(* CoDeSys 2.3 project: drillMachine_v5_WithPackML.pro *)
(* Title: Use of different IEC-61131-3 languages *)
(* Version: 1.0.0 *)
(* Author: Niko Siltala (TUT) *)
(* Description: Use of different IEC-61131-3 languages to control a lift door. *)
(* Libraries: Util.lib 29.1.20 23:45:11, STANDARD.LIB 16.8.17 14:08:57 *)

(* Global variable list: Global_Variables *)
VAR_GLOBAL
	(*Math constants*)
	MATH 				: CONSTANTS_MATH;		(*Mathematical constants from OSCAT 333*)
	lastRandom			: REAL;		(*Last Random number*)

	(*ConveyourIn - Left*)
	I_ConvIn_PartPresent: BOOL;	(*Sensor: Part is present*)
	O_ConvIn_MotON		: BOOL;	(*Conveyour In: Motor ON*)

	(*ConveyourOut - Right*)
	I_ConvOut_PartPresent: BOOL;(*Sensor: Part is present*)
	O_ConvOut_MotON		: BOOL;	(*Conveyour Out: Motor ON*)

	(*Manipulator - Left*)
	I_ManiL_Limit_Up	: BOOL;	(*Manipulator Left: Limit: Up*)
	I_ManiL_Limit_Dn	: BOOL;	(*Manipulator Left: Limit: Down*)
	I_ManiL_Limit_Home	: BOOL;	(*Manipulator Left: Home sensor*)
	I_ManiL_Turned_Left	: BOOL;	(*Manipulator Left: Turned to left*)
	I_ManiL_Turned_Right: BOOL;	(*Manipulator Left: Turned to right*)
	I_ManiL_Gripper_Open: BOOL;	(*Manipulator Left: Gripper is open*)

	O_ManiL_Turn_Left	: BOOL;	(*Manipulator Left: Turn to left position. Controls the valve*)
	O_ManiL_Turn_Right	: BOOL;	(*Manipulator Left: Turn to right position. Controls the valve*)
	O_ManiL_Gripper_Close: BOOL;(*Manipulator Left: Closes Gripper. Controls the valve*)

	bManiL_axZ_Enable	: BOOL;	(*Manipulator Left: Z-axis: enable*)
	bManiL_axZ_Start	: BOOL;	(*Manipulator Left: Z-axis: Start motion*)
	fManiL_axZ_Velo		: REAL;	(*Manipulator Left: Z-axis: Velocity*)
	fManiL_axZ_TargetPos: REAL;	(*Manipulator Left: Z-axis: Target position*)
	fManiL_axZ_CurrPos	: REAL;	(*Manipulator Left: Z-axis: Current position*)
	bManiL_axZ_InTargetPos	: BOOL;	(*Manipulator Left: Z-axis: Target position is reached*)

	(*Drilling Machine*)
	I_Drill_Limit_Up	: BOOL;	(*Drill: Limit: Up*)
	I_Drill_Limit_Dn	: BOOL;	(*Drill: Limit: Down*)
	I_Drill_Limit_Home	: BOOL;	(*Drill: Home sensor*)
	I_Drill_Fixture_Open: BOOL;	(*Drill: Fixture is open*)
	I_Drill_Fixture_Closed: BOOL;	(*Drill: Fixture is closed*)

	O_Drill_Spindle_On	: BOOL;	(*Drill: Turn on drill spindle.*)
	O_Drill_Fixture_Close: BOOL;(*Drill: Closes Fixture. Controls the valve*)

	bDrill_axZ_Enable	: BOOL;	(*Drill: Z-axis: enable*)
	bDrill_axZ_Start	: BOOL;	(*Drill: Z-axis: Start motion*)
	fDrill_axZ_Velo		: REAL;	(*Drill: Z-axis: Velocity*)
	fDrill_axZ_TargetPos: REAL;	(*Drill: Z-axis: Target position*)
	fDrill_axZ_CurrPos	: REAL;	(*Drill: Z-axis: Current position*)
	bDrill_axZ_InTargetPos	: BOOL;	(*Drill: Z-axis: Target position is reached*)

	(*Manipulator - Right*)
	I_ManiR_Limit_Up	: BOOL;	(*Manipulator Right: Limit: Up*)
	I_ManiR_Limit_Dn	: BOOL;	(*Manipulator Right: Limit: Down*)
	I_ManiR_Limit_Home	: BOOL;	(*Manipulator Right: Home sensor*)
	I_ManiR_Turned_Left	: BOOL;	(*Manipulator Right: Turned to left*)
	I_ManiR_Turned_Right: BOOL;	(*Manipulator Right: Turned to right*)
	I_ManiR_Gripper_Open: BOOL;	(*Manipulator Right: Gripper is open*)

	O_ManiR_Turn_Left	: BOOL;	(*Manipulator Right: Turn to left position. Controls the valve*)
	O_ManiR_Turn_Right	: BOOL;	(*Manipulator Right: Turn to right position. Controls the valve*)
	O_ManiR_Gripper_Close: BOOL;(*Manipulator Right: Closes Gripper. Controls the valve*)

	bManiR_axZ_Enable	: BOOL;	(*Manipulator Right: Z-axis: enable*)
	bManiR_axZ_Start	: BOOL;	(*Manipulator Right: Z-axis: Start motion*)
	fManiR_axZ_Velo		: REAL;	(*Manipulator Right: Z-axis: Velocity*)
	fManiR_axZ_TargetPos: REAL;	(*Manipulator Right: Z-axis: Target position*)
	fManiR_axZ_CurrPos	: REAL;	(*Manipulator Right: Z-axis: Current position*)
	bManiR_axZ_InTargetPos	: BOOL;	(*Manipulator Right: Z-axis: Target position is reached*)


	(*Control panel and indications*)
	I_EmergencyClear	: BOOL;	(*Emergency Circuit is clear*)
	I_Btn_Reset		: BOOL;	(*Button: Reset*)
	I_Btn_Start		: BOOL;	(*Button: Start*)
	I_Btn_Stop		: BOOL;	(*Button: Stop*)

	O_Light_Start	: BOOL;	(*Light: Running*)
	O_Light_Stop	: BOOL;	(*Light: Stopped*)
	O_Beacon_Red	: BOOL;	(*Beacon Light: red*)
	O_Beacon_Yellow	: BOOL;	(*Beacon Light: yellow*)
	O_Beacon_Green	: BOOL;	(*Beacon Light: green*)

(* -------------HMI INPUTS (from HMI to PLC) -------------------*)
	HMI_uModeReq		: UINT :=1;		(*Mode request. DEFAULT:PRODUCTION1*)
(* -------------HMI OUTPUTS (from PLC to HMI) -------------------*)
	PLC_uModeCurrent	: UINT;			(*Current Mode*)
	PLC_uStateCurrent	: UINT;			(*Current State*)

(*-----------------------FUNCTION BLOCKS----------------*)
	fbStateModel		: FB_PackMLStateModel_ST;	(*FB for executing PackML state model*)
END_VAR

(* Data type *)
TYPE CONSTANTS_MATH :
STRUCT
	PI : REAL := 	3.14159265358979323846264338327950288;		(* Kreiszahl PI *)
	PI2 : REAL := 	6.28318530717958647692528676655900576;	(* PI * 2 *)
	PI4 : REAL :=  12.56637061435917295385057353311801152;	(* PI * 4 *)
	PI05 : REAL :=  1.5707963267949;							(* PI / 2 *)
	PI025 : REAL := 0.785398163397448;							(* PI / 4 *)
	PI_INV : REAL := 0.318309886183791;						(* 1 / PI *)
	E : REAL := 	2.71828182845904523536028747135266249;		(* Euler constant e *)
	E_INV : REAL := 0.367879441171442;							(* 1 / e *)
	SQ2 : REAL :=	1.4142135623731;							(* Wurzel von 2 *)
	FACTS : ARRAY[0..12] OF DINT := 1,1,2,6,24,120,720,5040,40320,362880,3628800,39916800,479001600;
END_STRUCT
END_TYPE



(*
From OSCAT 333
revision history
hm	26.10.2008	rev 1.0
	original version

hm	26. mar. 2011	rev 1.1
	added array facts
*)

(* Data type *)
TYPE E_Mode :
(*UserModes: Modes for different production states*)
(
	eMode_undefined := 0,
	eMode_Automatic :=1,
	eMode_Manual :=3,
	eMode_Production1 :=5,
	eMode_Production2 :=6
);
END_TYPE

(* Data type *)
TYPE E_ModeProc :
(*Procedural control modes. Can be changed in any state*)
(
	eModeProc_undefined := 0,
	eModeProc_Automatic :=1,
	eModeProc_SemiAutomatic :=2,
	eModeProc_Manual :=3
);
END_TYPE

(* Data type *)
TYPE E_PackMLState :
(*PackML States*)
(
	eSt_Aborting :=0,
	eSt_Aborted,
	eSt_Clearing,
	eSt_Stopped,
	eSt_Stopping,
	eSt_Resetting,
	eSt_Idle,
	eSt_Starting,
	eSt_Execute,
	eSt_Suspending,
	eSt_Suspended,
	eSt_Unsuspending,
	eSt_Holding,
	eSt_Held,
	eSt_UnHolding,
	eSt_Completing,
	eSt_Completed
);
END_TYPE

(* Data type *)
TYPE EN_Mode :
	(eMode_Unknown := 0,
	eMode_Auto := 1,
	eMode_Manual );
END_TYPE

(* Data type *)
TYPE ST_Part :
(*Data structure for the simulated parts *)
STRUCT
	bExists		: BOOL;	(* Part exists *)
	bHasHole	: BOOL;	(* Part has hole *)
	posX		: REAL;	(* X-position of the part*)
	posY		: REAL;	(* Y-position of the part*)
END_STRUCT
END_TYPE

(* POU PRG/PRG_Blinking, ST *)
PROGRAM PRG_Blinking
(*Avustavia laskentaoperaatioita
- vilkutussignaalit
Author: Niko Siltala, niko.siltala@tut.fi, Tampere University of Technology / MEI
Date: 2016-12-12
Version: 1.0
*)
VAR_OUTPUT
	bSign4Hz:BOOL;					(*4 Hz (240krt/min) taajudella vaihteleva signaali*)
	bSign2Hz:BOOL;					(*2 Hz (120krt/min) taajudella vaihteleva signaali*)
	bSign1Hz:BOOL;					(*1 Hz (60krt/min) taajudella vaihteleva signaali*)
	bSign0_5Hz:BOOL;				(*0,5 Hz (30krt/min) taajudella vaihteleva signaali*)
END_VAR
VAR
	bInitDone	: BOOL	:=FALSE;	(*Ohjelman initialisointi*)
	TP_Delay:TP;				(*Nopein taajuus / 2 tuottaja*)
	bBaseHz:BOOL:=FALSE;		(*Nopein taajuus/2*)
	iBaseHz:UINT:=4;				(*Base taajuus (Hz)*)
	(*RTRIG_BASE: R_TRIG;		(*Base signaali nousee*)*)
	RTRIG_2Hz_Sign : R_TRIG;		(*2Hz signaalin generointi*)
	RTRIG_1Hz_Sign : R_TRIG;		(*1Hz signaalin generointi*)
	RTRIG_0_5Hz_Sign : R_TRIG;	(*0,5Hz signaalin generointi*)
	tBaseTaajuus:TIME;			(*Base vilkutuksen timerin arvo. f/2*)
	fPLC_CYCLE_TIME: LREAL;	(*PLC:n cycli aika. Sekunttia*)

END_VAR
(*Ohjelman initialisoinnit - Suoritetaan vain kertaalleen*)
IF NOT bInitDone THEN
	(*fPLC_CYCLE_TIME := UDINT_TO_LREAL(SystemTaskInfoArr[1].cycleTime) / 10E6; (*[s]*)*)
	fPLC_Cycle_Time := 1;	(*[s]*)
	(*Base Vilkkusignaalien tuottaminen*)
	(* 250ms - 1* cykliaika(20ms)*)
	tBaseTaajuus := LREAL_TO_TIME( ( (1/ UINT_TO_LREAL(iBaseHz) / 2 ) - 1 * fPLC_CYCLE_TIME ) * 1000);
	bInitDone := TRUE;
END_IF;

(*Base signaalin genrointi*)
TP_Delay(IN:=NOT TP_Delay.Q , PT:=tBaseTaajuus);
IF NOT TP_Delay.Q THEN
	bBaseHz := NOT bBaseHz;
	bSign4Hz:= bBaseHz;
END_IF;

(*2Hz signaalin genrointi*)
RTRIG_2Hz_Sign(CLK:=bSign4Hz);
IF RTRIG_2Hz_Sign.Q THEN
	bSign2Hz:=NOT bSign2Hz;
END_IF;

(*1Hz signaalin genrointi*)
RTRIG_1Hz_Sign(CLK:=bSign2Hz);
IF RTRIG_1Hz_Sign.Q THEN
	bSign1Hz:=NOT bSign1Hz;
END_IF;

(*0,5 Hz signaalin generointi*)
RTRIG_0_5Hz_Sign(CLK:=bSign1Hz);
IF (RTRIG_0_5Hz_Sign.Q) THEN
	bSign0_5Hz:= NOT bSign0_5Hz;
END_IF;
END_PROGRAM

(* POU PRG/PRG_ConveyorL, ST *)
PROGRAM PRG_ConveyorL
VAR_INPUT
	(* PackML Inputs *)
	State							: E_PackMLState;
	ControlMode					: E_Mode;
	ProceeduralMode				: E_ModeProc;

	hiPartAvail_FromLeft			: BOOL;
	hiRdyToReceive_FromRight  : BOOL;
END_VAR
VAR_OUTPUT
	(* PackML Outputs *)
	SC								: BOOL;
	bInitDone						: BOOL;
	bStopOk						: BOOL;
	bSuspend						: BOOL;

	hoReadyToRecieve_ToLeft	: BOOL;
	hoPartAvail_ToRight			: BOOL;
END_VAR
VAR
	initOK							: BOOL := FALSE;
	fbConveyorLeft				: FB_Conveyor_Left;
END_VAR
SC := FALSE;

CASE State OF
	eSt_Aborting:
		O_ConvIn_MotON		:= FALSE;
		SC 					:= TRUE;
	eSt_Clearing:
		SC 					:= TRUE;
	eSt_Resetting:
		SC 					:= TRUE;
	eSt_Starting:
		SC 					:= TRUE;
	;
	eSt_Holding:
	;
	eSt_UnHolding:
	;
	eSt_Suspending:
		fbConveyorLeft (I_Enable :=  FALSE);
		actUpdateIO;
		IF fbConveyorLeft.bStopOk THEN
			SC := TRUE;
		END_IF
	;
	eSt_Suspended:
		actUpdateIO;
		IF NOT fbConveyorLeft.bSuspend THEN
			bSuspend := FALSE;
		END_IF

	eSt_Unsuspending:
		SC := TRUE;
	eSt_Execute:
		CASE ControlMode OF
			eMode_Automatic:
				fbConveyorLeft (I_Enable	:= TRUE ,	I_Reset := FALSE );
				actUpdateIO;
				IF fbConveyorLeft.bSuspend THEN
					bSuspend := TRUE;
				ELSE
					bSuspend := FALSE;
				END_IF
			eMode_Manual:
			;
		END_CASE
		eSt_Completing:
		;

		eSt_Stopping:
			fbConveyorLeft (I_Enable :=  FALSE);
			actUpdateIO;
			IF fbConveyorLeft.bStopOk THEN
				bStopOk := TRUE;
				SC 	   := TRUE;
			ELSE
				bStopOk := FALSE;
			END_IF
END_CASE
END_PROGRAM
ACTION actUpdateIO:
fbConveyorLeft (
	I_PartEndSensor				:=  I_ConvIn_PartPresent,
	O_ConvRunning				=> O_ConvIn_MotON,
	hiPartAvail_FromLeft			:= hiPartAvail_FromLeft ,
	hiRdyToReceive_FromRight	:= hiRdyToReceive_FromRight,
	hoPartAvail_toRight			=> hoPartAvail_ToRight ,
	hoReadyToRecieve_ToLeft	=> hoReadyToRecieve_ToLeft );
END_ACTION

(* POU FBs/FB_Conveyor_Left, SFC *)
FUNCTION_BLOCK FB_Conveyor_Left
VAR_INPUT
	(* PackML Inputs *)
	State							: E_PackMLState;
	ControlMode					: E_Mode;
	ProceeduralMode				: E_ModeProc;

	I_Enable		 				: BOOL;
	I_Reset		 				: BOOL;
	I_PartEndSensor 				: BOOL;

	(* SMEMA Handshake Inputs *)
	hiPartAvail_FromLeft			: BOOL;
	hiRdyToReceive_FromRight	: BOOL;
END_VAR
VAR_OUTPUT
	(* PackML Outputs *)
	SC								: BOOL;

	(* SMEMA Handshake Outputs *)
	hoReadyToRecieve_ToLeft	: BOOL;
	hoPartAvail_ToRight			: BOOL;

	bInitialised					: BOOL;
	O_ConvRunning			       : BOOL;
	bStopOk						: BOOL;
	bSuspend						: BOOL;

END_VAR
VAR
	tonSuspendDelay			: TON;
	tSuspendDelay			: TIME := T#5s;
	bStartTrans				: BOOL := FALSE;
	bStopTrans				: BOOL := FALSE;
	bTranFinished			: BOOL := FALSE;
	bMachineReady			: BOOL := FALSE;
	bLocalReset				: BOOL := FALSE;	(*Performs local reset*)
	SFCReset 				: BOOL := FALSE;	(*Resets the execution of SFC to init once this SFCFlag is set true *)
END_VAR
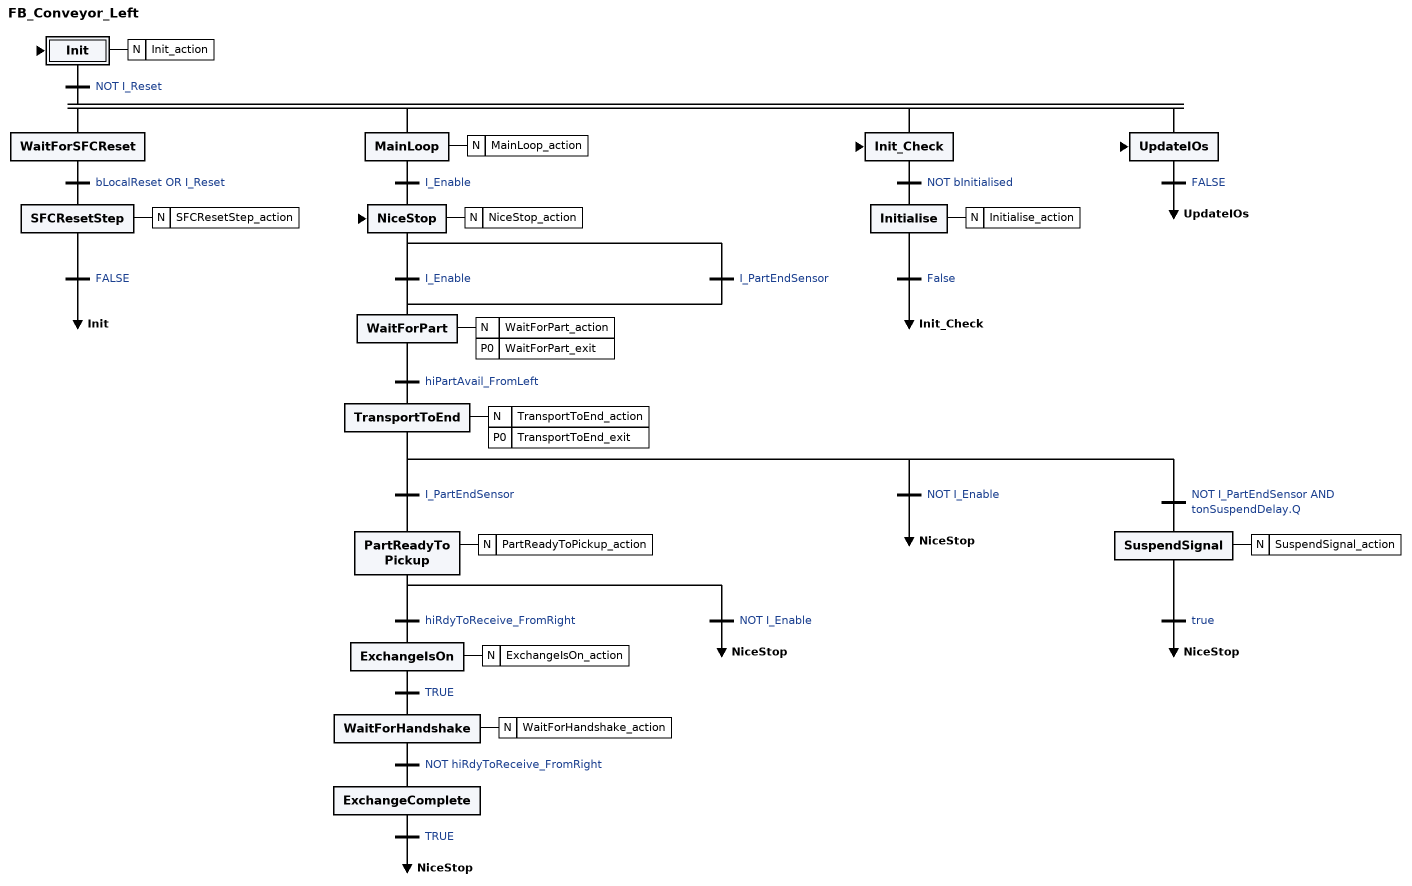
INITIAL_STEP Init:
	Init_action(N);
END_STEP
TRANSITION FROM Init TO (WaitForSFCReset, MainLoop, Init_Check, UpdateIOs) := NOT I_Reset;
END_TRANSITION
STEP WaitForSFCReset:
END_STEP
TRANSITION FROM WaitForSFCReset TO SFCResetStep := bLocalReset OR I_Reset;
END_TRANSITION
STEP MainLoop:
	MainLoop_action(N);
END_STEP
TRANSITION FROM MainLoop TO NiceStop := I_Enable;
END_TRANSITION
STEP Init_Check:
END_STEP
TRANSITION FROM Init_Check TO Initialise := NOT bInitialised;
END_TRANSITION
STEP Initialise:
	Initialise_action(N);
END_STEP
TRANSITION FROM Initialise TO Init_Check := False;
END_TRANSITION
STEP NiceStop:
	NiceStop_action(N);
END_STEP
TRANSITION FROM NiceStop TO WaitForPart := I_Enable;
END_TRANSITION
TRANSITION FROM NiceStop TO WaitForPart := I_PartEndSensor;
END_TRANSITION
STEP WaitForPart:
	WaitForPart_action(N);
	WaitForPart_exit(P0);
END_STEP
TRANSITION FROM WaitForPart TO TransportToEnd := hiPartAvail_FromLeft;
END_TRANSITION
STEP TransportToEnd:
	TransportToEnd_action(N);
	TransportToEnd_exit(P0);
END_STEP
TRANSITION FROM TransportToEnd TO PartReadyToPickup := I_PartEndSensor;
END_TRANSITION
TRANSITION FROM TransportToEnd TO NiceStop := NOT I_Enable;
END_TRANSITION
TRANSITION FROM TransportToEnd TO SuspendSignal := NOT I_PartEndSensor AND tonSuspendDelay.Q;
END_TRANSITION
STEP SuspendSignal:
	SuspendSignal_action(N);
END_STEP
TRANSITION FROM SuspendSignal TO NiceStop := true;
END_TRANSITION
STEP PartReadyToPickup:
	PartReadyToPickup_action(N);
END_STEP
TRANSITION FROM PartReadyToPickup TO ExchangeIsOn := hiRdyToReceive_FromRight;
END_TRANSITION
TRANSITION FROM PartReadyToPickup TO NiceStop := NOT I_Enable;
END_TRANSITION
STEP ExchangeIsOn:
	ExchangeIsOn_action(N);
END_STEP
TRANSITION FROM ExchangeIsOn TO WaitForHandshake := TRUE;
END_TRANSITION
STEP WaitForHandshake:
	WaitForHandshake_action(N);
END_STEP
TRANSITION FROM WaitForHandshake TO ExchangeComplete := NOT hiRdyToReceive_FromRight;
END_TRANSITION
STEP ExchangeComplete:
END_STEP
TRANSITION FROM ExchangeComplete TO NiceStop := TRUE;
END_TRANSITION
STEP UpdateIOs:
END_STEP
TRANSITION FROM UpdateIOs TO UpdateIOs := FALSE;
END_TRANSITION
STEP SFCResetStep:
	SFCResetStep_action(N);
END_STEP
TRANSITION FROM SFCResetStep TO Init := FALSE;
END_TRANSITION

ACTION Init_action:
SFCReset 		:= FALSE;
bLocalReset		:= FALSE;
O_ConvRunning	:= FALSE;
bStopOk 			:= TRUE;
bInitialised		:= FALSE;
bSuspend	 		:= FALSE;
END_ACTION

ACTION MainLoop_action:
hoPartAvail_toRight := FALSE;
END_ACTION

ACTION Initialise_action:
bInitialised := TRUE;
END_ACTION

ACTION NiceStop_action:
bStopOk := TRUE;
O_ConvRunning := TRUE;
hoPartAvail_ToRight := FALSE;
END_ACTION

ACTION WaitForPart_action:
hoReadyToRecieve_ToLeft := TRUE;
bSuspend	 := FALSE;
END_ACTION

ACTION WaitForPart_exit:
bStopOk := FALSE;
END_ACTION

ACTION TransportToEnd_action:
O_ConvRunning := TRUE;
tonSuspendDelay(IN:=TRUE , PT:= tSuspendDelay);
END_ACTION

ACTION TransportToEnd_exit:
tonSuspendDelay(IN:=FALSE);
END_ACTION

ACTION SuspendSignal_action:
bSuspend := TRUE;
END_ACTION

ACTION PartReadyToPickup_action:
hoPartAvail_ToRight := TRUE;
END_ACTION

ACTION ExchangeIsOn_action:
hoReadyToRecieve_ToLeft := FALSE;
END_ACTION

ACTION WaitForHandshake_action:
hoPartAvail_ToRight := FALSE;
END_ACTION

ACTION SFCResetStep_action:
SFCReset := TRUE;
END_ACTION
END_FUNCTION_BLOCK

(* POU PRG/PRG_ConveyorR, ST *)
PROGRAM PRG_ConveyorR
VAR_INPUT
	(* PackML Inputs *)
	State							: E_PackMLState;
	ControlMode					: E_Mode;
	ProceeduralMode				: E_ModeProc;

	hiPartAvail_FromLeft			: BOOL;
	hiRdyToReceive_FromRight  : BOOL;
END_VAR
VAR_OUTPUT
	(* PackML Outputs *)
	SC								: BOOL;
	bInitDone						: BOOL;
	bStopOk						: BOOL;

	hoReadyToRecieve_ToLeft	: BOOL;
	hoPartAvail_ToRight			: BOOL;
END_VAR
VAR
	initOK							: BOOL := FALSE;
	fbConveyorRight				: FB_Conveyor_Right;
END_VAR
SC := FALSE;

CASE State OF
	eSt_Aborting:
		O_ConvOut_MotON		:= FALSE;
		SC := TRUE;
	eSt_Clearing:
		SC := TRUE;
	eSt_Resetting:
		SC := TRUE;
	eSt_Starting:
		SC  := TRUE;
	eSt_Holding:
	;
	eSt_UnHolding:
	;
	eSt_Suspending:
		fbConveyorRight (I_Enable :=  FALSE);
		actUpdateIO;
		IF fbConveyorRight.bStopOk THEN
			SC := TRUE;
		END_IF
	eSt_Unsuspending:
		SC := TRUE;
	eSt_Execute:
		CASE ControlMode OF
			eMode_Automatic:
				fbConveyorRight (I_Enable := TRUE , I_Reset := FALSE );
				actUpdateIO;
			eMode_Manual:
			;
		END_CASE
	eSt_Completing:
	;

	eSt_Stopping:
		fbConveyorRight (I_Enable :=  FALSE);
		actUpdateIO;
		IF fbConveyorRight.bStopOk THEN
			bStopOk := TRUE;
			SC 	   := TRUE;
		ELSE
			bStopOk := FALSE;
			END_IF
END_CASE
END_PROGRAM
ACTION actUpdateIO:
fbConveyorRight (
	I_PartEndSensor				:=  I_ConvOut_PartPresent,
	O_ConvRunning				=> O_ConvOut_MotON,
	hiPartAvail_FromLeft			:= hiPartAvail_FromLeft ,
	hiRdyToReceive_FromRight	:= hiRdyToReceive_FromRight,
	hoPartAvail_toRight			=> hoPartAvail_ToRight ,
	hoReadyToRecieve_ToLeft	=> hoReadyToRecieve_ToLeft );
END_ACTION

(* POU FBs/FB_Conveyor_Right, SFC *)
FUNCTION_BLOCK FB_Conveyor_Right
VAR_INPUT
	(* PackML Inputs *)
	State							: E_PackMLState;
	ControlMode					: E_Mode;
	ProceeduralMode				: E_ModeProc;

	I_Enable		 				: BOOL;
	I_Reset		 				: BOOL;
	I_PartEndSensor 				: BOOL;

	(* SMEMA Handshake Inputs *)
	hiPartAvail_FromLeft			: BOOL;
	hiRdyToReceive_FromRight	: BOOL;
END_VAR
VAR_OUTPUT
	(* PackML Outputs *)
	SC								: BOOL;

	(* SMEMA Handshake Outputs *)
	hoReadyToRecieve_ToLeft	: BOOL;
	hoPartAvail_ToRight			: BOOL;
	O_ConvRunning			       : BOOL;
	bInitialised					: BOOL;
	bStopOk						: BOOL;


END_VAR
VAR
	bStartTrans				: BOOL := FALSE;
	bStopTrans				: BOOL := FALSE;
	bTranFinished			: BOOL := FALSE;
	bMachineReady			: BOOL := FALSE;
	bLocalReset				: BOOL := FALSE;	(*Performs local reset*)
	SFCReset 				: BOOL := FALSE;	(*Resets the execution of SFC to init once this SFCFlag is set true *)
	I_Sensor_PartInsideMachine: BOOL;
END_VAR
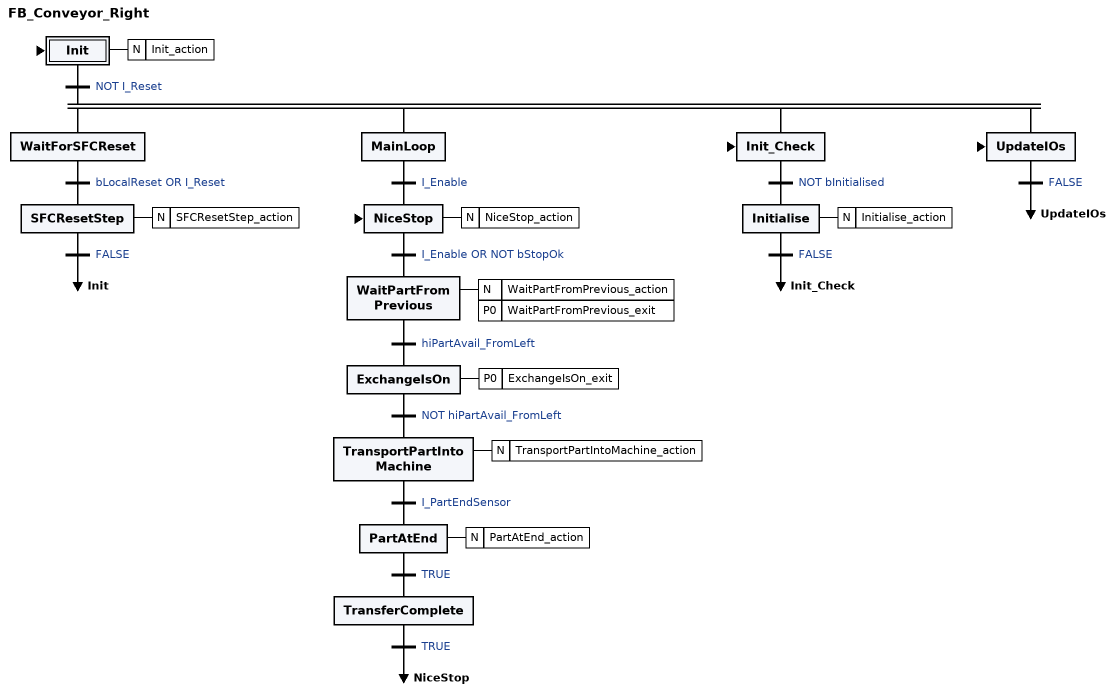
INITIAL_STEP Init:
	Init_action(N);
END_STEP
TRANSITION FROM Init TO (WaitForSFCReset, MainLoop, Init_Check, UpdateIOs) := NOT I_Reset;
END_TRANSITION
STEP WaitForSFCReset:
END_STEP
TRANSITION FROM WaitForSFCReset TO SFCResetStep := bLocalReset OR I_Reset;
END_TRANSITION
STEP MainLoop:
END_STEP
TRANSITION FROM MainLoop TO NiceStop := I_Enable;
END_TRANSITION
STEP Init_Check:
END_STEP
TRANSITION FROM Init_Check TO Initialise := NOT bInitialised;
END_TRANSITION
STEP Initialise:
	Initialise_action(N);
END_STEP
TRANSITION FROM Initialise TO Init_Check := FALSE;
END_TRANSITION
STEP NiceStop:
	NiceStop_action(N);
END_STEP
TRANSITION FROM NiceStop TO WaitPartFromPrevious := I_Enable OR NOT bStopOk;
END_TRANSITION
STEP WaitPartFromPrevious:
	WaitPartFromPrevious_action(N);
	WaitPartFromPrevious_exit(P0);
END_STEP
TRANSITION FROM WaitPartFromPrevious TO ExchangeIsOn := hiPartAvail_FromLeft;
END_TRANSITION
STEP ExchangeIsOn:
	ExchangeIsOn_exit(P0);
END_STEP
TRANSITION FROM ExchangeIsOn TO TransportPartIntoMachine := NOT hiPartAvail_FromLeft;
END_TRANSITION
STEP TransportPartIntoMachine:
	TransportPartIntoMachine_action(N);
END_STEP
TRANSITION FROM TransportPartIntoMachine TO PartAtEnd := I_PartEndSensor;
END_TRANSITION
STEP PartAtEnd:
	PartAtEnd_action(N);
END_STEP
TRANSITION FROM PartAtEnd TO TransferComplete := TRUE;
END_TRANSITION
STEP TransferComplete:
END_STEP
TRANSITION FROM TransferComplete TO NiceStop := TRUE;
END_TRANSITION
STEP UpdateIOs:
END_STEP
TRANSITION FROM UpdateIOs TO UpdateIOs := FALSE;
END_TRANSITION
STEP SFCResetStep:
	SFCResetStep_action(N);
END_STEP
TRANSITION FROM SFCResetStep TO Init := FALSE;
END_TRANSITION

ACTION Init_action:
SFCReset := FALSE;
bLocalReset	:= FALSE;
O_ConvRunning := FALSE;
bStopOK	 := TRUE;
bInitialised := FALSE;
END_ACTION

ACTION Initialise_action:
bInitialised := TRUE;
END_ACTION

ACTION NiceStop_action:
IF hiPartAvail_FromLeft THEN
	bStopOk := FALSE;
ELSE
	bStopOk := TRUE;
END_IF
END_ACTION

ACTION WaitPartFromPrevious_action:
hoReadyToRecieve_ToLeft := TRUE;
hoPartAvail_toRight := FALSE;
END_ACTION

ACTION WaitPartFromPrevious_exit:
bStopOK	:= FALSE;
END_ACTION

ACTION ExchangeIsOn_exit:
O_ConvRunning := FALSE;
END_ACTION

ACTION TransportPartIntoMachine_action:
O_ConvRunning := TRUE;
hoReadyToRecieve_ToLeft := FALSE;
END_ACTION

ACTION PartAtEnd_action:
O_ConvRunning := FALSE;
hoPartAvail_ToRight := TRUE;
END_ACTION

ACTION SFCResetStep_action:
SFCReset := TRUE;
END_ACTION
END_FUNCTION_BLOCK

(* POU PRG/PRG_Drill, ST *)
PROGRAM PRG_Drill
VAR_INPUT
	(* PackML Inputs *)
	State							: E_PackMLState;
	ControlMode					: E_Mode;
	ProceeduralMode				: E_ModeProc;

	hiPartAvail_FromLeft			: BOOL;
	hiRdyToReceive_FromRight  : BOOL;
END_VAR
VAR_OUTPUT
	(* PackML Outputs *)
	SC								: BOOL;
	bInitDone						: BOOL;
	bStopOk						: BOOL;

	hoReadyToRecieve_ToLeft	: BOOL;
	hoPartAvail_ToRight			: BOOL;
END_VAR
VAR
	fbDrill 							: FB_Drill;
END_VAR
SC := FALSE;

CASE State OF
	eSt_Aborting:
		bDrill_axZ_Start 					:= FALSE;
		O_Drill_Spindle_On				:= FALSE;
		(*  Avoid Toggling fixture Objects *)
		IF I_Drill_Fixture_Open THEN
			O_Drill_Fixture_Close 		:= FALSE;
		ELSE
			O_Drill_Fixture_Close		:= TRUE;
		END_IF
		SC := TRUE;
	eSt_Clearing:
		SC := TRUE;
	eSt_Resetting:
		SC := TRUE;
	eSt_Starting:
		IF NOT  fbDrill.bInitialised THEN
			actUpdateIO;
		ELSE
			bInitDone	 := TRUE;
			SC		 := TRUE;
		END_IF

	;
	eSt_Holding:
	;
	eSt_UnHolding:
	;
	eSt_Suspending:
		fbDrill (I_Enable :=  FALSE);
		actUpdateIO;
		IF fbDrill.bStopOk THEN
			SC := TRUE;
		END_IF
	eSt_Unsuspending:
		SC := TRUE;
	eSt_Execute:
		CASE ControlMode OF
			eMode_Automatic:
				fbDrill (
					I_Enable						:= TRUE,
					I_Reset						:= FALSE);
				actUpdateIO;
			eMode_Manual:
			;
		END_CASE
		eSt_Completing:
		;

		eSt_Stopping:
			fbDrill (I_Enable :=  FALSE);
			actUpdateIO;
			IF fbDrill.bStopOk THEN
				bStopOk := TRUE;
				SC 	   := TRUE;
			ELSE
				bStopOk := FALSE;
			END_IF
END_CASE
END_PROGRAM
ACTION actUpdateIO:
fbDrill (
	I_Drill_Limit_Up				:= I_Drill_Limit_Up,
	I_Drill_Limit_Dn				:= I_Drill_Limit_Dn ,
	I_Drill_Limit_Home			:= I_Drill_Limit_Home,
	I_Drill_Fixture_Open			:= I_Drill_Fixture_Open,
	I_Drill_Fixture_Closed		:= I_Drill_Fixture_Closed,
	fDrill_axZ_CurrPos			:= fDrill_axZ_CurrPos ,
	bDrill_axZ_InTargetPos		:= bDrill_axZ_InTargetPos ,

	hiPartAvail_FromLeft			:= hiPartAvail_FromLeft ,
	hiRdyToReceive_FromRight	:= hiRdyToReceive_FromRight ,
	hoReadyToRecieve_ToLeft	=>hoReadyToRecieve_ToLeft ,
	hoPartAvail_ToRight			=>hoPartAvail_ToRight ,

	O_Drill_Spindle_On			=> O_Drill_Spindle_On ,
	O_Drill_Fixture_Close		=> O_Drill_Fixture_Close ,
	bDrill_axZ_Enable			=> bDrill_axZ_Enable ,
	bDrill_axZ_Start				=> bDrill_axZ_Start ,
	fDrill_axZ_Velo				=> fDrill_axZ_Velo,
	fDrill_axZ_TargetPos			=> fDrill_axZ_TargetPos );
END_ACTION

(* POU FBs/FB_Drill, SFC *)
FUNCTION_BLOCK FB_Drill
VAR_INPUT
	(* PackML Inputs *)
	State							: E_PackMLState;
	ControlMode					: E_Mode;
	ProceeduralMode				: E_ModeProc;

	I_Enable		 				: BOOL;
	I_Reset		 				: BOOL;
	I_StopRequest				: BOOL;

	(* SMEMA HandshakeInputs *)
	hiPartAvail_FromLeft			: BOOL;
	hiRdyToReceive_FromRight	: BOOL;

	(* Drill Sensor *)
	I_Drill_Limit_Up				: BOOL;	(*Drill: Limit: Up*)
	I_Drill_Limit_Dn				: BOOL;	(*Drill: Limit: Down*)
	I_Drill_Limit_Home			: BOOL;	(*Drill: Home sensor*)
	I_Drill_Fixture_Open			: BOOL;	(*Drill: Fixture is open*)
	I_Drill_Fixture_Closed		: BOOL;	(*Drill: Fixture is closed*)

	(* Drill Inputs Controls *)
	fDrill_axZ_CurrPos			: REAL;	(*Drill: Z-axis: Current position*)
	bDrill_axZ_InTargetPos		: BOOL;	(*Drill: Z-axis: Target position is reached*)
END_VAR
VAR_OUTPUT
	(* PackML Outputs *)
	SC								: BOOL;

	O_Drill_Spindle_On			: BOOL;	(*Drill: Turn on drill spindle.*)
	O_Drill_Fixture_Close		: BOOL;	(*Drill: Closes Fixture. Controls the valve*)
	bInitialised					: BOOL;
	bStopOk						: BOOL;

	(* SMEMA HandshakeInputs *)
	hoReadyToRecieve_ToLeft	: BOOL;
	hoPartAvail_ToRight			: BOOL;

	(* Drill Outputs *)
	bDrill_axZ_Enable			: BOOL;	(*Drill: Z-axis: enable*)
	bDrill_axZ_Start				: BOOL;	(*Drill: Z-axis: Start motion*)
	fDrill_axZ_Velo				: REAL;	(*Drill: Z-axis: Velocity*)
	fDrill_axZ_TargetPos			: REAL;	(*Drill: Z-axis: Target position*)

END_VAR
VAR

	bDrillHomed				: BOOL := FALSE;
	bStartCycle				: BOOL := FALSE;
	bLocalReset				: BOOL := FALSE;	(*Performs local reset*)
	SFCReset 				: BOOL := FALSE;	(*Resets the execution of SFC to init once this SFCFlag is set true *)
	tonMoveDelay				: TON;
	tMoveDelay				: TIME := T#1s;
	bDrill						: BOOL;
	bDrilled					: BOOL;

END_VAR
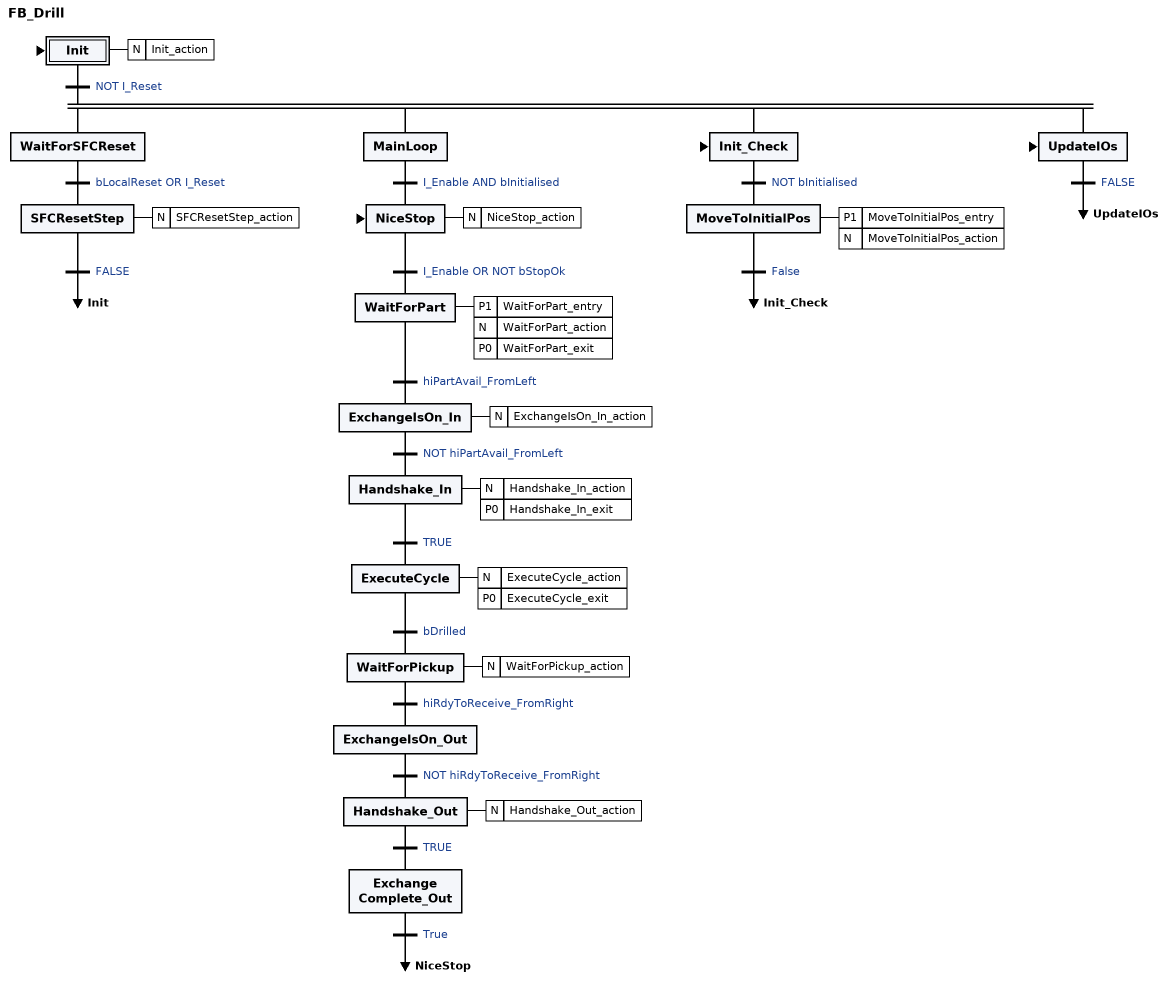
INITIAL_STEP Init:
	Init_action(N);
END_STEP
TRANSITION FROM Init TO (WaitForSFCReset, MainLoop, Init_Check, UpdateIOs) := NOT I_Reset;
END_TRANSITION
STEP WaitForSFCReset:
END_STEP
TRANSITION FROM WaitForSFCReset TO SFCResetStep := bLocalReset OR I_Reset;
END_TRANSITION
STEP MainLoop:
END_STEP
TRANSITION FROM MainLoop TO NiceStop := I_Enable AND bInitialised;
END_TRANSITION
STEP Init_Check:
END_STEP
TRANSITION FROM Init_Check TO MoveToInitialPos := NOT bInitialised;
END_TRANSITION
STEP MoveToInitialPos:
	MoveToInitialPos_entry(P1);
	MoveToInitialPos_action(N);
END_STEP
TRANSITION FROM MoveToInitialPos TO Init_Check := False;
END_TRANSITION
STEP NiceStop:
	NiceStop_action(N);
END_STEP
TRANSITION FROM NiceStop TO WaitForPart := I_Enable OR NOT bStopOk;
END_TRANSITION
STEP WaitForPart:
	WaitForPart_entry(P1);
	WaitForPart_action(N);
	WaitForPart_exit(P0);
END_STEP
TRANSITION FROM WaitForPart TO ExchangeIsOn_In := hiPartAvail_FromLeft;
END_TRANSITION
STEP ExchangeIsOn_In:
	ExchangeIsOn_In_action(N);
END_STEP
TRANSITION FROM ExchangeIsOn_In TO Handshake_In := NOT hiPartAvail_FromLeft;
END_TRANSITION
STEP Handshake_In:
	Handshake_In_action(N);
	Handshake_In_exit(P0);
END_STEP
TRANSITION FROM Handshake_In TO ExecuteCycle := TRUE;
END_TRANSITION
STEP ExecuteCycle:
	ExecuteCycle_action(N);
	ExecuteCycle_exit(P0);
END_STEP
TRANSITION FROM ExecuteCycle TO WaitForPickup := bDrilled;
END_TRANSITION
STEP WaitForPickup:
	WaitForPickup_action(N);
END_STEP
TRANSITION FROM WaitForPickup TO ExchangeIsOn_Out := hiRdyToReceive_FromRight;
END_TRANSITION
STEP ExchangeIsOn_Out:
END_STEP
TRANSITION FROM ExchangeIsOn_Out TO Handshake_Out := NOT hiRdyToReceive_FromRight;
END_TRANSITION
STEP Handshake_Out:
	Handshake_Out_action(N);
END_STEP
TRANSITION FROM Handshake_Out TO ExchangeComplete_Out := TRUE;
END_TRANSITION
STEP ExchangeComplete_Out:
END_STEP
TRANSITION FROM ExchangeComplete_Out TO NiceStop := True;
END_TRANSITION
STEP UpdateIOs:
END_STEP
TRANSITION FROM UpdateIOs TO UpdateIOs := FALSE;
END_TRANSITION
STEP SFCResetStep:
	SFCResetStep_action(N);
END_STEP
TRANSITION FROM SFCResetStep TO Init := FALSE;
END_TRANSITION

ACTION Init_action:
(* Status Flags *)
bStopOK			:= TRUE;
bInitialised 		:= FALSE;
bDrillHomed 		:= FALSE;
(* Reset Flags *)
SFCReset 		:= FALSE;
bLocalReset		:= FALSE;
(* Handshake Flags*)
hoReadyToRecieve_ToLeft	:= FALSE;
hoPartAvail_ToRight			:= FALSE;
END_ACTION

ACTION MoveToInitialPos_entry:
bStopOk := FALSE;
END_ACTION

ACTION MoveToInitialPos_action:
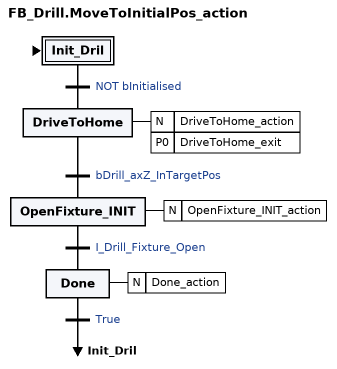
INITIAL_STEP Init_Dril:
END_STEP
TRANSITION FROM Init_Dril TO DriveToHome := NOT bInitialised;
END_TRANSITION
STEP DriveToHome:
	DriveToHome_action(N);
	DriveToHome_exit(P0);
END_STEP
TRANSITION FROM DriveToHome TO OpenFixture_INIT := bDrill_axZ_InTargetPos;
END_TRANSITION
STEP OpenFixture_INIT:
	OpenFixture_INIT_action(N);
END_STEP
TRANSITION FROM OpenFixture_INIT TO Done := I_Drill_Fixture_Open;
END_TRANSITION
STEP Done:
	Done_action(N);
END_STEP
TRANSITION FROM Done TO Init_Dril := True;
END_TRANSITION

ACTION DriveToHome_action:
bDrill_axZ_Enable		:= TRUE;
fDrill_axZ_TargetPos		:= -10;
fDrill_axZ_Velo			:= 5;
bDrill_axZ_Start			:= TRUE;
END_ACTION

ACTION DriveToHome_exit:
bDrill_axZ_Start := FALSE;
END_ACTION

ACTION OpenFixture_INIT_action:
O_Drill_Fixture_Close := FALSE;
END_ACTION

ACTION Done_action:
bInitialised := TRUE;
bStopOk := TRUE;
END_ACTION
END_ACTION

ACTION NiceStop_action:
IF hiPartAvail_FromLeft THEN
	bStopOk := FALSE;
ELSE
	bStopOk := TRUE;
END_IF
END_ACTION

ACTION WaitForPart_entry:
bStopOK	:= TRUE;
END_ACTION

ACTION WaitForPart_action:
hoReadyToRecieve_ToLeft := TRUE;
END_ACTION

ACTION WaitForPart_exit:
bStopOK	:= FALSE;
END_ACTION

ACTION ExchangeIsOn_In_action:
hoReadyToRecieve_ToLeft	:= TRUE;
END_ACTION

ACTION Handshake_In_action:
hoReadyToRecieve_ToLeft := FALSE;
END_ACTION

ACTION Handshake_In_exit:
bDrill := TRUE;
END_ACTION

ACTION ExecuteCycle_action:
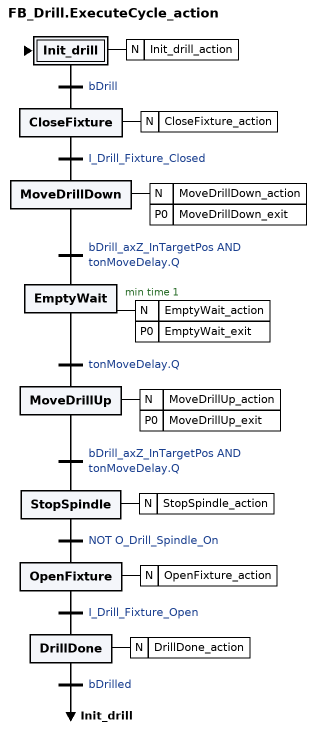
INITIAL_STEP Init_drill:
	Init_drill_action(N);
END_STEP
TRANSITION FROM Init_drill TO CloseFixture := bDrill;
END_TRANSITION
STEP CloseFixture:
	CloseFixture_action(N);
END_STEP
TRANSITION FROM CloseFixture TO MoveDrillDown := I_Drill_Fixture_Closed;
END_TRANSITION
STEP MoveDrillDown:
	MoveDrillDown_action(N);
	MoveDrillDown_exit(P0);
END_STEP
TRANSITION FROM MoveDrillDown TO EmptyWait := bDrill_axZ_InTargetPos AND tonMoveDelay.Q;
END_TRANSITION
STEP EmptyWait: (* min time 1 *)
	EmptyWait_action(N);
	EmptyWait_exit(P0);
END_STEP
TRANSITION FROM EmptyWait TO MoveDrillUp := tonMoveDelay.Q;
END_TRANSITION
STEP MoveDrillUp:
	MoveDrillUp_action(N);
	MoveDrillUp_exit(P0);
END_STEP
TRANSITION FROM MoveDrillUp TO StopSpindle := bDrill_axZ_InTargetPos AND tonMoveDelay.Q;
END_TRANSITION
STEP StopSpindle:
	StopSpindle_action(N);
END_STEP
TRANSITION FROM StopSpindle TO OpenFixture := NOT O_Drill_Spindle_On;
END_TRANSITION
STEP OpenFixture:
	OpenFixture_action(N);
END_STEP
TRANSITION FROM OpenFixture TO DrillDone := I_Drill_Fixture_Open;
END_TRANSITION
STEP DrillDone:
	DrillDone_action(N);
END_STEP
TRANSITION FROM DrillDone TO Init_drill := bDrilled;
END_TRANSITION

ACTION Init_drill_action:
O_Drill_Spindle_On	:= FALSE;
bDrill_axZ_Enable	:= FALSE;
bDrill_axZ_Start		:= FALSE;
fDrill_axZ_Velo		:= 0;
END_ACTION

ACTION CloseFixture_action:
bDrilled 					:= FALSE;
O_Drill_Fixture_Close 	:= TRUE;
END_ACTION

ACTION MoveDrillDown_action:
bDrill_axZ_Enable := TRUE;
fDrill_axZ_Velo :=10;
fDrill_axZ_TargetPos := -140;
bDrill_axZ_Start := TRUE;
tonMoveDelay(IN:=TRUE , PT:= tMoveDelay);
O_Drill_Spindle_On := TRUE;
END_ACTION

ACTION MoveDrillDown_exit:
bDrill_axZ_Start := FALSE;
tonMoveDelay(IN:=FALSE );
END_ACTION

ACTION EmptyWait_action:
tonMoveDelay(IN:=TRUE , PT:= tMoveDelay);
END_ACTION

ACTION EmptyWait_exit:
tonMoveDelay(IN:=FALSE);
END_ACTION

ACTION MoveDrillUp_action:
tonMoveDelay(IN:=TRUE , PT:= tMoveDelay);
fDrill_axZ_Velo :=10;
fDrill_axZ_TargetPos := -10;
bDrill_axZ_Start := TRUE;
END_ACTION

ACTION MoveDrillUp_exit:
bDrill_axZ_Start := FALSE;
tonMoveDelay(IN:=FALSE);
END_ACTION

ACTION StopSpindle_action:
O_Drill_Spindle_On := FALSE;
END_ACTION

ACTION OpenFixture_action:
O_Drill_Fixture_Close	:= FALSE;
END_ACTION

ACTION DrillDone_action:
bDrilled := TRUE;
bDrill := FALSE;
END_ACTION
END_ACTION

ACTION ExecuteCycle_exit:
bDrilled := FALSE;
END_ACTION

ACTION WaitForPickup_action:
hoPartAvail_ToRight := TRUE;
END_ACTION

ACTION Handshake_Out_action:
hoPartAvail_ToRight := FALSE;
END_ACTION

ACTION SFCResetStep_action:
SFCReset := TRUE;
END_ACTION
END_FUNCTION_BLOCK

(* POU PRG_MAIN_DRILL_MACHINE, ST *)
PROGRAM PRG_MAIN_DRILL_MACHINE
VAR
	(* PackML Related Variables *)
	bBlink					: BOOL;	(*1s blinkg for CodeSys Simulation*)
	c						: INT;	(*Support variable for blinking*)

	partCount				: R_TRIG;
	bAllOkToStop		       : BOOL := TRUE;
	bInit_FirstBoot			: BOOL := FALSE;
	bStopRequested		: BOOL := FALSE;
	bE_StopRestart		: BOOL := FALSE;
	oStopRequested		: BOOL;

	itemToProduce 		: INT := 1;
	itemProduced 		: INT := 0;

END_VAR
(* ****** Section 1: Initialisations and default values. Initial conditions for variables on every PLC cycle*)
fbStateModel.bSC := FALSE;
actCountParts;
actCheckOKtoStop;

(* ****** Section 2: Actions in your program without considering the Control Mode. I.e. actions are performed same way indenpendent on
current Control Mode selection.*)
(*Mode independent state actions*)
CASE fbStateModel.eState OF
eSt_Aborting:
	(* One can make specific actions in case of specific Mode-State combination.
	   One can also consider to call a specific program when in specific Mode-State combination*)
	(*actAborting;*)
	bInit_FirstBoot := FALSE;
	fbStateModel.bSC := PRG_ConveyorL.SC AND	PRG_ManipulatorLeft.SC  AND PRG_Drill.SC AND
						     PRG_ManipulatorRight.SC AND  PRG_ConveyorR.SC;
eSt_Clearing:
	fbStateModel.bSC := PRG_ConveyorL.SC AND PRG_ManipulatorLeft.SC  AND PRG_Drill.SC AND
						     PRG_ManipulatorRight.SC AND  PRG_ConveyorR.SC;
eSt_Stopping:
	fbStateModel.bSC := PRG_ConveyorL.SC AND PRG_ManipulatorLeft.SC  AND PRG_Drill.SC AND
						     PRG_ManipulatorRight.SC AND  PRG_ConveyorR.SC;
eSt_Resetting:
	fbStateModel.bSC := PRG_ConveyorL.SC AND PRG_ManipulatorLeft.SC  AND PRG_Drill.SC AND
						     PRG_ManipulatorRight.SC AND  PRG_ConveyorR.SC;
eSt_Holding:
	fbStateModel.bSC := TRUE;		(*TODO: Remove/Replace this row with desired actions*)
eSt_UnHolding:
	fbStateModel.bSC := TRUE;		(*TODO: Remove/Replace this row with desired actions*)
eSt_Suspending:
	fbStateModel.bSC := PRG_ConveyorL.SC AND PRG_ManipulatorLeft.SC  AND PRG_Drill.SC AND
						     PRG_ManipulatorRight.SC AND  PRG_ConveyorR.SC;
	;
	(*fbStateModel.bSC := TRUE; *)		(*TODO: Remove/Replace this row with desired actions*)
eSt_Unsuspending:
	fbStateModel.bSC := PRG_ConveyorL.SC AND PRG_ManipulatorLeft.SC  AND PRG_Drill.SC AND
						     PRG_ManipulatorRight.SC AND  PRG_ConveyorR.SC;
END_CASE;

(* ****** Section 3: Actions in your program which are Control Mode specific. Two nested case structures where outer one selects the
control mode and inner the PackML state. In order to avoid conflicts, it would be better to process each PackML state either in Section 2 
or Section 3, but not in both. *)
(*Execution mode related state actions*)
CASE fbStateModel.eMode OF
(*MODE: MANUAL*)
eMode_Manual:
	(* ****** Section 3.1: PackML state based processing actions when Control Mode is Manual.*)
	CASE fbStateModel.eState OF
	eSt_Idle:
		fbStateModel.bAck_Completed := FALSE;		(*TODO: Remove/Replace this row with desired actions*)
	eSt_Starting:
		fbStateModel.bSC := TRUE;					(*TODO: Remove/Replace this row with desired actions*)
	eSt_Completing:
		fbStateModel.bSC := TRUE;					(*TODO: Remove/Replace this row with desired actions*)
	eSt_Completed:
		fbStateModel.bAck_Completed := TRUE;		(*TODO: Remove/Replace this row with desired actions*)
	END_CASE;

(*MODE: AUTOMATIC*)
eMode_Automatic:
	(* ****** Section 3.2: PackML state based processing actions when Control Mode is Automatic.*)
	CASE fbStateModel.eState OF
	eSt_Idle:
		fbStateModel.bAck_Completed := FALSE;		(*TODO: Remove/Replace this row with desired actions*)
	eSt_Starting:
			fbStateModel.bSC := PRG_ConveyorL.SC AND PRG_ManipulatorLeft.SC  AND PRG_Drill.SC AND
						     		     PRG_ManipulatorRight.SC AND  PRG_ConveyorR.SC;
	eSt_Completing:
		fbStateModel.bSC := TRUE;					(*TODO: Remove/Replace this row with desired actions*)
	eSt_Completed:
		;
		(*fbStateModel.bAck_Completed:= I_Btn_Start;*)
	END_CASE;

(*MODE: UNKNOWN*)
ELSE	(*This is an Error branch.*)
	; (*TODO: Make implementation*)
END_CASE;

(* ****** Section 4: Grouping PackML states for calling Programs or FB instances.
This is to avoid repetition inside case structure in Section 3. With IF clause setting lower (and upper) state limits we can filter out the states when we want to call 
specific programs. The order of states is defined in Tab:Data types > E_PackMLState. eSt_Aborting is lowest and eSt_Completed is highest.
Here we filter calling programs, only when we are in higher states than Stopped. Inside IF there is again CASE which process each Control Mode separately.*)
(*Execution part. Making calls for program if we are on states above Stopped*)
IF (fbStateModel.eState > eSt_Stopped) THEN
	CASE fbStateModel.eMode OF
		(*MODE: MANUAL*)
		eMode_Manual:
			;
		(*MODE: AUTOMATIC*)
		eMode_Automatic:
			;
	END_CASE;
END_IF;

(* ****** Section 5: Calling the fbStateModel instance.
Here the instance of state model is called and all triggering inputs are set, but bSC (State Completed), which you control in your programs. 
This is indication that your program has  finished certain stage.
- Pay attention where the instance fbStateModel is defined. Do you do it in global variables or e.g. here in PRG_MAIN? Important is to use the 
same instance in all places, so that machine state is unique and shared. Remember, if you have multiple definitions, the PRG_MAIN "hides" 
the global one, and might lead to problems elswhere, when you think you are using the same instance, but actually are not. 
- In case you are using the PackML visualisation (VC_PackMLStates), make sure you connect its placeholder to the very same PackML FB instance.
- The Mask for wIgnoreState is created as following. I use binary base for the value(2#). The lowest bit in the mask corresponds the eSt_Aborting
 in E_PackMLState. The next is eSt_Aborted, and so on. Specific state is ignored and jumped over when it is masked out i.e. ignored by having 1 
in that position. Note that implementation allows this only for selected states. See FB_PackMLStateModel_ST code for further details.*)
(*Calling & Updating the state model*)
(*TODO: Evaluate and change all input conditions according your application needs*)
fbStateModel(
	bResetFB			:= ,
	eModeReq		:= HMI_uModeReq,
	wIgnoreState		:= 2#100000,		(*TODO: Which states should be ignodered. Default: 2#000000 or 2#100000*)
	bSC				:= ,		(*Must NOT be assigned ANY variable, because fb input is directly assigned above by your programs!!!*)
	bAbort				:= NOT I_EmergencyClear,
	bClear				:= I_EmergencyClear,
	bReset			:= ,
	bStart				:= I_Btn_Start,
	bHold				:= ,
	bUn_Hold			:= ,
	bSuspend			:= PRG_ConveyorL.bSuspend AND bAllOkToStop,
	bUn_Suspend	:= NOT PRG_ConveyorL.bSuspend,
	bStop				:= I_Btn_Stop,
	bComplete		:= ,
	bAck_Completed	:= ,
	eMode				=> ,
	eState				=> );

(* ****** Section 6: Here we update all outputs according the current state of our PackML model. This allows us to process the in single location.
The control of outputs is bind to state, not e.g. to inputs. The inputs are the one driving the PackML model forward. Again CASE structure can be used.*)
(*Call for HMI and UI update*)
HMI_and_UI_Update;


PRG_ConveyorL(
	State							:= fbStateModel.eState ,
	ControlMode					:= fbStateModel.eMode,
	ProceeduralMode				:= ,
	hiPartAvail_FromLeft			:= TRUE ,
	hiRdyToReceive_FromRight	:= PRG_ManipulatorLeft.hoReadyToRecieve_ToLeft,
	SC								=> ,
	bInitDone						=> ,
	bStopOk						=> ,
	hoReadyToRecieve_ToLeft	=> ,
	hoPartAvail_ToRight			=> );

PRG_ManipulatorLeft(
	State							:= fbStateModel.eState,
	ControlMode					:= fbStateModel.eMode ,
	ProceeduralMode				:= ,
	hiPartAvail_FromLeft			:= PRG_ConveyorL.hoPartAvail_ToRight ,
	hiRdyToReceive_FromRight	:= PRG_Drill.hoReadyToRecieve_ToLeft,
	SC								=> ,
	bInitDone						=> ,
	bStopOk						=> ,
	hoReadyToRecieve_ToLeft	=> ,
	hoPartAvail_ToRight			=> );

PRG_Drill(
	State							:= fbStateModel.eState,
	ControlMode					:= fbStateModel.eMode ,
	ProceeduralMode				:= ,
	hiPartAvail_FromLeft			:= PRG_ManipulatorLeft.hoPartAvail_ToRight ,
	hiRdyToReceive_FromRight	:= PRG_ManipulatorRight.hoReadyToRecieve_ToLeft,
	SC								=> ,
	bInitDone						=> ,
	bStopOk						=> ,
	hoReadyToRecieve_ToLeft	=> ,
	hoPartAvail_ToRight			=> );

PRG_ManipulatorRight(
	State							:= fbStateModel.eState ,
	ControlMode					:= fbStateModel.eMode ,
	ProceeduralMode				:= ,
	hiPartAvail_FromLeft			:= PRG_Drill.hoPartAvail_ToRight,
	hiRdyToReceive_FromRight	:= PRG_ConveyorR.hoReadyToRecieve_ToLeft,
	SC								=> ,
	bInitDone						=> ,
	bStopOk						=> ,
	hoReadyToRecieve_ToLeft	=> ,
	hoPartAvail_ToRight			=> );

PRG_ConveyorR(
	State							:= fbStateModel.eState ,
	ControlMode					:= fbStateModel.eMode,
	ProceeduralMode				:= ,
	hiPartAvail_FromLeft			:= PRG_ManipulatorRight.hoPartAvail_ToRight,
	hiRdyToReceive_FromRight	:= TRUE,
	SC								=> ,
	bInitDone						=> ,
	bStopOk						=> ,
	hoReadyToRecieve_ToLeft	=> ,
	hoPartAvail_ToRight			=> );
END_PROGRAM
ACTION actAborting:
(* Conveyors *)
O_ConvIn_MotON					:= FALSE;
O_ConvOut_MotON	 			:= FALSE;

(* Manipulators *)
O_ManiL_Turn_Left		 		:= FALSE;
O_ManiL_Turn_Right		 		:= FALSE;
O_ManiR_Turn_Left		 		:= FALSE;
O_ManiR_Turn_Right		 		:= FALSE;
bManiL_axZ_Start					:= FALSE;
bManiR_axZ_Start				:= FALSE;

(*  Avoid Dropping Objects *)
IF I_ManiL_Gripper_Open THEN
	O_ManiL_Gripper_Close 	:= FALSE;
ELSE
	O_ManiL_Gripper_Close		:= TRUE;
END_IF
(* Drill *)
bDrill_axZ_Start 					:= FALSE;
O_Drill_Spindle_On				:= FALSE;

(*  Avoid Toggling fixture Objects *)
IF I_Drill_Fixture_Open THEN
	O_Drill_Fixture_Close 		:= FALSE;
ELSE
	O_Drill_Fixture_Close		:= TRUE;
END_IF

(*
fbConveyorLeft(I_Reset:=TRUE, bRun := FALSE);
fbConveyorRight(I_Reset:=TRUE, bRun := FALSE);
fbManipulatorLeft(I_Reset:=TRUE, I_Enable := FALSE);
fbManipulatorRight(I_Reset:=TRUE, I_Enable := FALSE);
fbDrill(I_Reset:=TRUE, I_Enable := FALSE);
*)
END_ACTION
ACTION actCheckOkToStop:
IF PRG_ConveyorL.bStopOk  AND PRG_ManipulatorLeft.bStopOk  AND PRG_Drill.bStopOk AND PRG_ManipulatorRight.bStopOk AND  PRG_ConveyorR.bStopOk THEN
	bAllOkToStop := TRUE;
ELSE
	bAllOkToStop := FALSE;
END_IF
END_ACTION
ACTION actCountParts:
partCount(CLK:= I_ConvOut_PartPresent, Q=> );
IF partCount.Q THEN
	itemProduced := itemProduced + 1;
END_IF
END_ACTION
ACTION HMI_and_UI_Update:
(*HMI Update*)
(*Calling blinking sub-program*)
PRG_Blinking (bSign4Hz=> , bSign2Hz=> , bSign1Hz=> , bSign0_5Hz=> );
(*Codesys simulation 1Hz blinking *)
c:= c + 1;
IF c > 1 THEN
	c:=0;
END_IF;
bBlink := (c=0);	(*bBlink is true if c=0*)

(*Init values*)
O_Light_Stop := FALSE;	(*TODO: Change initial values according your app needs*)

(*TODO: Change values according range of states *)
(*Start light*)
O_Light_Start :=  (fbStateModel.eState > eSt_Idle) AND (fbStateModel.eState < eSt_Completed);
IF (fbStateModel.eState > eSt_Completing) OR (fbStateModel.eState <= eSt_Execute) THEN
	O_Beacon_Yellow := FALSE;
END_IF

CASE fbStateModel.eState OF
eSt_Aborting, eSt_Aborted,eSt_Clearing:
	O_Light_Stop 		 := bBlink;
	O_Beacon_Red 	 := bBlink;
	O_Light_Start 		 := FALSE;
	O_Beacon_Green := FALSE;
eSt_Stopping, eSt_Stopped, eSt_Completed:
	O_Beacon_Green:= FALSE;
	IF  fbStateModel.eState = eSt_Stopping THEN
		O_Beacon_Green:= bBlink;
		O_Light_Start 		:= bBlink;
	END_IF
	O_Light_Stop 		:= TRUE;
	O_Beacon_Red 	:= TRUE;
eSt_Starting:
	O_Light_Start 		:= bBlink;
	O_Light_Stop 		 := FALSE;
	O_Beacon_Green:= bBlink;
	O_Beacon_Red 	 := FALSE;
eSt_Suspended, eSt_Suspending, eSt_Held:
	O_Light_Start 		 := bBlink;
	O_Beacon_Green	 := bBlink;
	O_Beacon_Yellow := TRUE;
	O_Beacon_Red 	 := FALSE;
eSt_Execute:
	O_Beacon_Red 	 := FALSE;
	O_Beacon_Green	 := TRUE;
END_CASE;
END_ACTION

(* POU PRG/PRG_ManipulatorLeft, ST *)
PROGRAM PRG_ManipulatorLeft
VAR_INPUT
	(* PackML Inputs *)
	State							: E_PackMLState;
	ControlMode					: E_Mode;
	ProceeduralMode				: E_ModeProc;

	hiPartAvail_FromLeft			: BOOL;
	hiRdyToReceive_FromRight  : BOOL;
END_VAR
VAR_OUTPUT
	(* PackML Outputs *)
	SC								: BOOL;
	bInitDone						: BOOL;
	bStopOk						: BOOL;

	hoReadyToRecieve_ToLeft	: BOOL;
	hoPartAvail_ToRight			: BOOL;
END_VAR
VAR
	initOK							: BOOL := FALSE;
	fbManipulatorLeft 				: FB_Manipulator;
END_VAR
SC := FALSE;

CASE State OF
	eSt_Aborting:
		O_ManiL_Turn_Left		 		:= FALSE;
		O_ManiL_Turn_Right		 		:= FALSE;
		bManiL_axZ_Start					:= FALSE;
		IF I_ManiL_Gripper_Open THEN
			O_ManiL_Gripper_Close 	:= FALSE;
		ELSE
			O_ManiL_Gripper_Close		:= TRUE;
		END_IF
		SC := TRUE;
	eSt_Clearing:
		SC := TRUE;
	;
	eSt_Resetting:
		SC := TRUE
	;

	eSt_Starting:
		IF NOT  fbManipulatorLeft.bInitialised THEN
			actUpdateIO;
		ELSE
			bInitDone	:= TRUE;
			SC		 	:= TRUE;
		END_IF
	;
	eSt_Holding:
	;
	eSt_UnHolding:
	;
	eSt_Suspending:
		fbManipulatorLeft (I_Enable :=  FALSE);
		actUpdateIO;
		IF fbManipulatorLeft.bStopOk THEN
			SC := TRUE;
		END_IF
	eSt_Unsuspending:
		SC := TRUE;
	eSt_Execute:
		CASE ControlMode OF
			eMode_Automatic:
				fbManipulatorLeft (
					I_Enable						:=  TRUE,
					b_LeftManip					:=  TRUE );
				actUpdateIO;

			eMode_Manual:
			;
		END_CASE
		eSt_Completing:
		;
	
		eSt_Stopping:
			fbManipulatorLeft (I_Enable :=  FALSE);
			actUpdateIO;
			IF fbManipulatorLeft.bStopOk THEN
				bStopOk := TRUE;
				SC 	   := TRUE;
			ELSE
				bStopOk := FALSE;
			END_IF
END_CASE
END_PROGRAM
ACTION actUpdateIO:
fbManipulatorLeft (
					b_LeftManip					:= TRUE ,
					I_Mani_Limit_Up				:= I_ManiL_Limit_Up,
					I_Mani_Limit_Dn				:= I_ManiL_Limit_Dn,
					I_Mani_Limit_Home			:= I_ManiL_Limit_Home ,
					I_Mani_Turned_Left			:= I_ManiL_Turned_Left,
					I_Mani_Turned_Right			:= I_ManiL_Turned_Right ,
					I_Mani_Gripper_Open		:= I_ManiL_Gripper_Open ,
					I_fMani_axZ_CurrPos			:= fManiL_axZ_CurrPos ,
					I_bMani_axZ_InTargetPos	:= bManiL_axZ_InTargetPos,

					hiPartAvail_FromLeft			:= hiPartAvail_FromLeft ,
					hiRdyToReceive_FromRight	:= hiRdyToReceive_FromRight,
					hoReadyToRecieve_ToLeft	=> hoReadyToRecieve_ToLeft,
					hoPartAvail_ToRight			=> hoPartAvail_ToRight ,
			
					O_Mani_Turn_Left			=> O_ManiL_Turn_Left ,
					O_Mani_Turn_Right			=> O_ManiL_Turn_Right ,
					O_Mani_Gripper_Close		=> O_ManiL_Gripper_Close ,
					O_bMani_axZ_Enable		=> bManiL_axZ_Enable ,
					O_bMani_axZ_Start			=> bManiL_axZ_Start ,
					O_fMani_axZ_Velo			=> fManiL_axZ_Velo,
					O_fMani_axZ_TargetPos		=> fManiL_axZ_TargetPos );
END_ACTION

(* POU FBs/FB_Manipulator, SFC *)
FUNCTION_BLOCK FB_Manipulator
VAR_INPUT
	(* PackML Inputs *)
	State							: E_PackMLState;
	ControlMode					: E_Mode;
	ProceeduralMode				: E_ModeProc;

	I_Enable		 				: BOOL;
	I_Reset		 				: BOOL;
	b_LeftManip					: BOOL;
	I_StopRequest				: BOOL;

	(* SMEMA HandshakeInputs *)
	hiPartAvail_FromLeft			: BOOL;
	hiRdyToReceive_FromRight	: BOOL;

	(* Manipulator Sensor *)
	I_Mani_Limit_Up				: BOOL;	(*Manipulator Left: Limit: Up*)
	I_Mani_Limit_Dn				: BOOL;	(*Manipulator Left: Limit: Down*)
	I_Mani_Limit_Home			: BOOL;	(*Manipulator Left: Home sensor*)
	I_Mani_Turned_Left			: BOOL;	(*Manipulator Left: Turned to left*)
	I_Mani_Turned_Right			: BOOL;	(*Manipulator Left: Turned to right*)
	I_Mani_Gripper_Open		: BOOL;	(*Manipulator Left: Gripper is open*)

	(* Manipulator Controls *)
	I_fMani_axZ_CurrPos			: REAL;	(*Manipulator Left: Z-axis: Current position*)
	I_bMani_axZ_InTargetPos	: BOOL;	(*Manipulator Left: Z-axis: Target position is reached*)

END_VAR
VAR_OUTPUT
	(* PackML Outputs *)
	SC								: BOOL;
	bInitialised					: BOOL;
	bStopOk						: BOOL;

	(* SMEMA Handshake Outputs *)
	hoReadyToRecieve_ToLeft	: BOOL;
	hoPartAvail_ToRight			: BOOL;

	(* Manipulator Outputs *)
	O_Mani_Turn_Left			: BOOL;	(*Manipulator Left: Turn to left position. Controls the valve*)
	O_Mani_Turn_Right			: BOOL;	(*Manipulator Left: Turn to right position. Controls the valve*)
	O_Mani_Gripper_Close		: BOOL;(*Manipulator Left: Closes Gripper. Controls the valve*)

	(* Manipulator Z axis Control *)
	O_bMani_axZ_Enable		: BOOL;	(*Manipulator Left: Z-axis: enable*)
	O_bMani_axZ_Start			: BOOL;	(*Manipulator Left: Z-axis: Start motion*)
	O_fMani_axZ_Velo			: REAL;	(*Manipulator Left: Z-axis: Velocity*)
	O_fMani_axZ_TargetPos		: REAL;	(*Manipulator Left: Z-axis: Target position*)


END_VAR
VAR
	bPick						: BOOL := FALSE;
	bPicked					: BOOL := FALSE;
	bPlace						: BOOL := FALSE;
	bPlaced					: BOOL := FALSE;
	bManipulatorHomed		: BOOL := FALSE;

	bLocalReset				: BOOL := FALSE;	(*Performs local reset*)
	SFCReset 				: BOOL := FALSE;	(*Resets the execution of SFC to init once this SFCFlag is set true *)
	tonMoveDelay				: TON;
	tMoveDelay				: TIME := T#1s;
	tHomeDelay				: TIME := T#700ms;

END_VAR
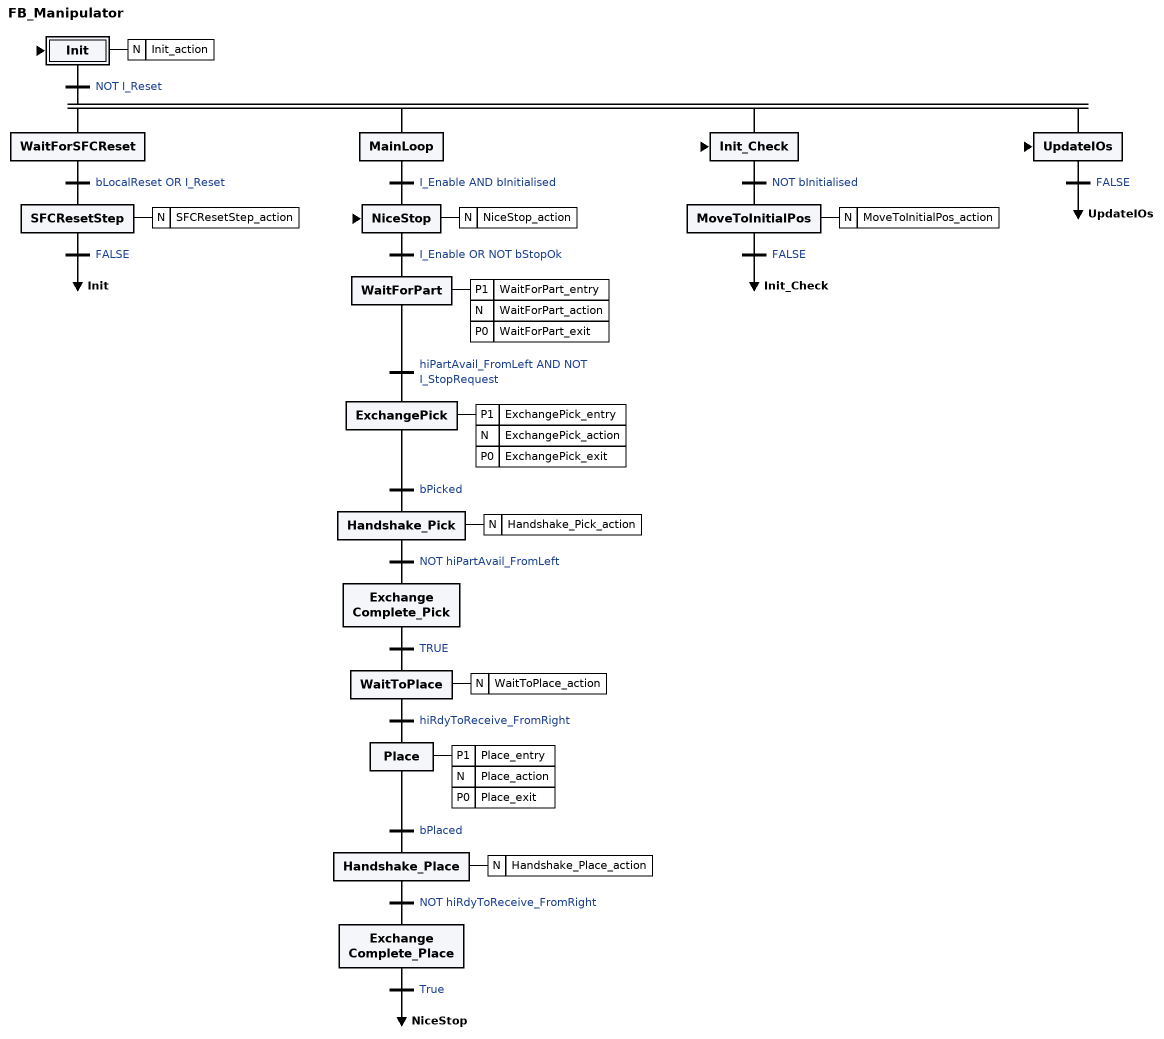
INITIAL_STEP Init:
	Init_action(N);
END_STEP
TRANSITION FROM Init TO (WaitForSFCReset, MainLoop, Init_Check, UpdateIOs) := NOT I_Reset;
END_TRANSITION
STEP WaitForSFCReset:
END_STEP
TRANSITION FROM WaitForSFCReset TO SFCResetStep := bLocalReset OR I_Reset;
END_TRANSITION
STEP MainLoop:
END_STEP
TRANSITION FROM MainLoop TO NiceStop := I_Enable AND bInitialised;
END_TRANSITION
STEP Init_Check:
END_STEP
TRANSITION FROM Init_Check TO MoveToInitialPos := NOT bInitialised;
END_TRANSITION
STEP MoveToInitialPos:
	MoveToInitialPos_action(N);
END_STEP
TRANSITION FROM MoveToInitialPos TO Init_Check := FALSE;
END_TRANSITION
STEP NiceStop:
	NiceStop_action(N);
END_STEP
TRANSITION FROM NiceStop TO WaitForPart := I_Enable OR NOT bStopOk;
END_TRANSITION
STEP WaitForPart:
	WaitForPart_entry(P1);
	WaitForPart_action(N);
	WaitForPart_exit(P0);
END_STEP
TRANSITION FROM WaitForPart TO ExchangePick := hiPartAvail_FromLeft AND NOT I_StopRequest;
END_TRANSITION
STEP ExchangePick:
	ExchangePick_entry(P1);
	ExchangePick_action(N);
	ExchangePick_exit(P0);
END_STEP
TRANSITION FROM ExchangePick TO Handshake_Pick := bPicked;
END_TRANSITION
STEP Handshake_Pick:
	Handshake_Pick_action(N);
END_STEP
TRANSITION FROM Handshake_Pick TO ExchangeComplete_Pick := NOT hiPartAvail_FromLeft;
END_TRANSITION
STEP ExchangeComplete_Pick:
END_STEP
TRANSITION FROM ExchangeComplete_Pick TO WaitToPlace := TRUE;
END_TRANSITION
STEP WaitToPlace:
	WaitToPlace_action(N);
END_STEP
TRANSITION FROM WaitToPlace TO Place := hiRdyToReceive_FromRight;
END_TRANSITION
STEP Place:
	Place_entry(P1);
	Place_action(N);
	Place_exit(P0);
END_STEP
TRANSITION FROM Place TO Handshake_Place := bPlaced;
END_TRANSITION
STEP Handshake_Place:
	Handshake_Place_action(N);
END_STEP
TRANSITION FROM Handshake_Place TO ExchangeComplete_Place := NOT hiRdyToReceive_FromRight;
END_TRANSITION
STEP ExchangeComplete_Place:
END_STEP
TRANSITION FROM ExchangeComplete_Place TO NiceStop := True;
END_TRANSITION
STEP UpdateIOs:
END_STEP
TRANSITION FROM UpdateIOs TO UpdateIOs := FALSE;
END_TRANSITION
STEP SFCResetStep:
	SFCResetStep_action(N);
END_STEP
TRANSITION FROM SFCResetStep TO Init := FALSE;
END_TRANSITION

ACTION Init_action:
(* State Flags *)
bManipulatorHomed 			:= FALSE;
bStopOK						:= TRUE;
bInitialised					:= FALSE;

(* Reset Flags *)
SFCReset 					:= FALSE;
bLocalReset					:= FALSE;

(* Init Handshakes *)
hoReadyToRecieve_ToLeft	:= FALSE;
hoPartAvail_ToRight			:= FALSE;
END_ACTION

ACTION MoveToInitialPos_action:
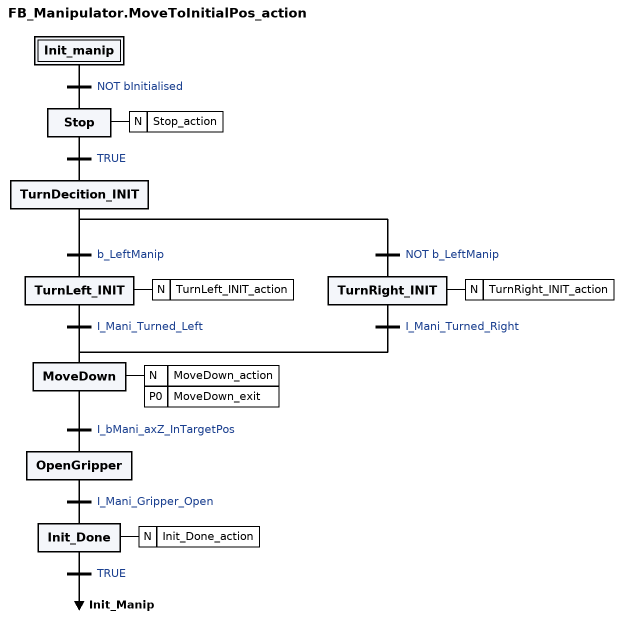
INITIAL_STEP Init_manip:
END_STEP
TRANSITION FROM Init_manip TO Stop := NOT bInitialised;
END_TRANSITION
STEP Stop:
	Stop_action(N);
END_STEP
TRANSITION FROM Stop TO TurnDecition_INIT := TRUE;
END_TRANSITION
STEP TurnDecition_INIT:
END_STEP
TRANSITION FROM TurnDecition_INIT TO TurnLeft_INIT := b_LeftManip;
END_TRANSITION
TRANSITION FROM TurnDecition_INIT TO TurnRight_INIT := NOT b_LeftManip;
END_TRANSITION
STEP TurnLeft_INIT:
	TurnLeft_INIT_action(N);
END_STEP
TRANSITION FROM TurnLeft_INIT TO MoveDown := I_Mani_Turned_Left;
END_TRANSITION
STEP TurnRight_INIT:
	TurnRight_INIT_action(N);
END_STEP
TRANSITION FROM TurnRight_INIT TO MoveDown := I_Mani_Turned_Right;
END_TRANSITION
STEP MoveDown:
	MoveDown_action(N);
	MoveDown_exit(P0);
END_STEP
TRANSITION FROM MoveDown TO OpenGripper := I_bMani_axZ_InTargetPos;
END_TRANSITION
STEP OpenGripper:
END_STEP
TRANSITION FROM OpenGripper TO Init_Done := I_Mani_Gripper_Open;
END_TRANSITION
STEP Init_Done:
	Init_Done_action(N);
END_STEP
TRANSITION FROM Init_Done TO Init_Manip := TRUE;
END_TRANSITION

ACTION Stop_action:
O_fMani_axZ_Velo		:= 0;
O_Mani_Turn_Left		:= FALSE;
O_Mani_Turn_Right		:= FALSE;
END_ACTION

ACTION TurnLeft_INIT_action:
O_Mani_Turn_Right 	 := FALSE;
O_Mani_Turn_Left 	 := TRUE;
END_ACTION

ACTION TurnRight_INIT_action:
O_Mani_Turn_Right 	 := TRUE;
O_Mani_Turn_Left 	 := FALSE;
END_ACTION

ACTION MoveDown_action:
O_bMani_axZ_Enable		:= TRUE;
tonMoveDelay(IN:=TRUE , PT:= tMoveDelay);
O_fMani_axZ_Velo			:= 5;
O_fMani_axZ_TargetPos		:= -45;
O_bMani_axZ_Start			:= TRUE;
END_ACTION

ACTION MoveDown_exit:
tonMoveDelay(IN:=FALSE);
END_ACTION

ACTION Init_Done_action:
bInitialised := TRUE;
END_ACTION
END_ACTION

ACTION NiceStop_action:
IF hiPartAvail_FromLeft THEN
	bStopOk := FALSE;
ELSE
	bStopOk := TRUE;
END_IF
END_ACTION

ACTION WaitForPart_entry:
bPicked := FALSE;
bPlaced := FALSE;
END_ACTION

ACTION WaitForPart_action:
hoReadyToRecieve_ToLeft	 := TRUE;
END_ACTION

ACTION WaitForPart_exit:
bStopOK	:= FALSE;
END_ACTION

ACTION ExchangePick_entry:
bPick := TRUE;
END_ACTION

ACTION ExchangePick_action:
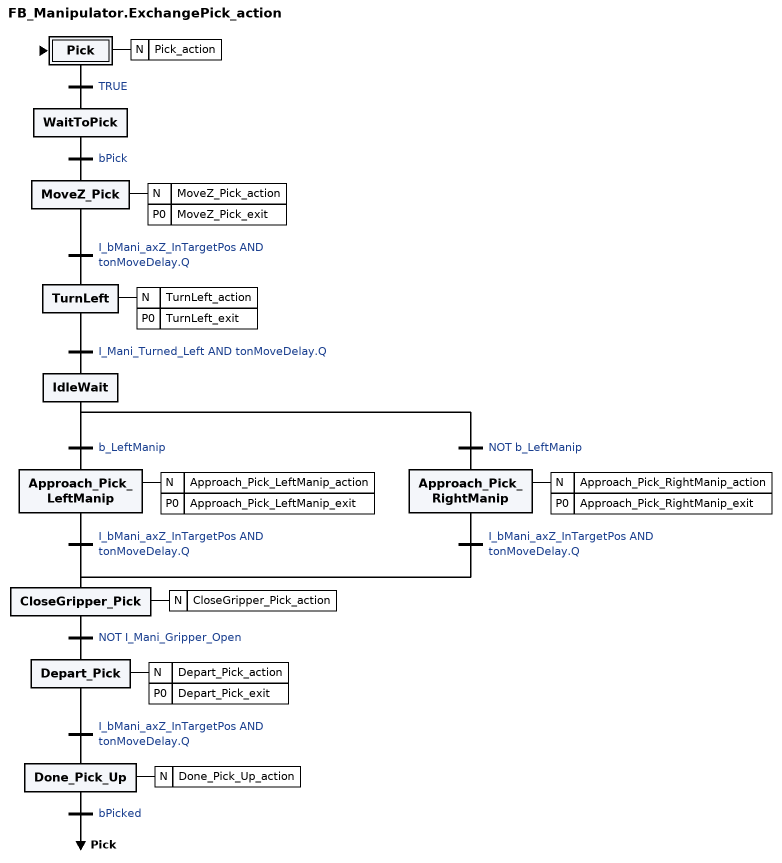
INITIAL_STEP Pick:
	Pick_action(N);
END_STEP
TRANSITION FROM Pick TO WaitToPick := TRUE;
END_TRANSITION
STEP WaitToPick:
END_STEP
TRANSITION FROM WaitToPick TO MoveZ_Pick := bPick;
END_TRANSITION
STEP MoveZ_Pick:
	MoveZ_Pick_action(N);
	MoveZ_Pick_exit(P0);
END_STEP
TRANSITION FROM MoveZ_Pick TO TurnLeft := I_bMani_axZ_InTargetPos AND tonMoveDelay.Q;
END_TRANSITION
STEP TurnLeft:
	TurnLeft_action(N);
	TurnLeft_exit(P0);
END_STEP
TRANSITION FROM TurnLeft TO IdleWait := I_Mani_Turned_Left AND tonMoveDelay.Q;
END_TRANSITION
STEP IdleWait:
END_STEP
TRANSITION FROM IdleWait TO Approach_Pick_LeftManip := b_LeftManip;
END_TRANSITION
TRANSITION FROM IdleWait TO Approach_Pick_RightManip := NOT b_LeftManip;
END_TRANSITION
STEP Approach_Pick_LeftManip:
	Approach_Pick_LeftManip_action(N);
	Approach_Pick_LeftManip_exit(P0);
END_STEP
TRANSITION FROM Approach_Pick_LeftManip TO CloseGripper_Pick := I_bMani_axZ_InTargetPos AND tonMoveDelay.Q;
END_TRANSITION
STEP Approach_Pick_RightManip:
	Approach_Pick_RightManip_action(N);
	Approach_Pick_RightManip_exit(P0);
END_STEP
TRANSITION FROM Approach_Pick_RightManip TO CloseGripper_Pick := I_bMani_axZ_InTargetPos AND tonMoveDelay.Q;
END_TRANSITION
STEP CloseGripper_Pick:
	CloseGripper_Pick_action(N);
END_STEP
TRANSITION FROM CloseGripper_Pick TO Depart_Pick := NOT I_Mani_Gripper_Open;
END_TRANSITION
STEP Depart_Pick:
	Depart_Pick_action(N);
	Depart_Pick_exit(P0);
END_STEP
TRANSITION FROM Depart_Pick TO Done_Pick_Up := I_bMani_axZ_InTargetPos AND tonMoveDelay.Q;
END_TRANSITION
STEP Done_Pick_Up:
	Done_Pick_Up_action(N);
END_STEP
TRANSITION FROM Done_Pick_Up TO Pick := bPicked;
END_TRANSITION

ACTION Pick_action:
bPicked := FALSE;
END_ACTION

ACTION MoveZ_Pick_action:
O_bMani_axZ_Enable := TRUE;
tonMoveDelay(IN:=TRUE , PT:= tMoveDelay);
O_fMani_axZ_Velo :=10;
O_fMani_axZ_TargetPos := -45;
O_bMani_axZ_Start := TRUE;
END_ACTION

ACTION MoveZ_Pick_exit:
tonMoveDelay(IN:=FALSE );
O_bMani_axZ_Start := FALSE;
END_ACTION

ACTION TurnLeft_action:
tonMoveDelay(IN:=TRUE , PT:= tMoveDelay);
O_Mani_Turn_Left 	 := TRUE;
O_Mani_Turn_Right 	 := FALSE;
END_ACTION

ACTION TurnLeft_exit:
tonMoveDelay(IN:=FALSE);
END_ACTION

ACTION Approach_Pick_LeftManip_action:
bPicked := FALSE;
tonMoveDelay(IN:=TRUE , PT:= tMoveDelay);
O_fMani_axZ_Velo :=10;
O_fMani_axZ_TargetPos := -120;
O_bMani_axZ_Start := TRUE;
END_ACTION

ACTION Approach_Pick_LeftManip_exit:
O_bMani_axZ_Start := FALSE;
tonMoveDelay(IN:=FALSE);
END_ACTION

ACTION Approach_Pick_RightManip_action:
bPicked := FALSE;
tonMoveDelay(IN:=TRUE , PT:= tMoveDelay);
O_fMani_axZ_Velo :=10;
O_fMani_axZ_TargetPos := -74;
O_bMani_axZ_Start := TRUE;
END_ACTION

ACTION Approach_Pick_RightManip_exit:
O_bMani_axZ_Start := FALSE;
tonMoveDelay(IN:=FALSE);
END_ACTION

ACTION CloseGripper_Pick_action:
O_Mani_Gripper_Close := TRUE;
END_ACTION

ACTION Depart_Pick_action:
O_fMani_axZ_Velo :=10;
O_fMani_axZ_TargetPos := -45;
O_bMani_axZ_Start := TRUE;
tonMoveDelay(IN:=TRUE , PT:= tMoveDelay);
END_ACTION

ACTION Depart_Pick_exit:
O_bMani_axZ_Start := FALSE;
tonMoveDelay(IN:=FALSE);
END_ACTION

ACTION Done_Pick_Up_action:
bPick		 := FALSE;
bPicked	 := TRUE;
END_ACTION
END_ACTION

ACTION ExchangePick_exit:
bPick := FALSE;
bPlaced := FALSE;
END_ACTION

ACTION Handshake_Pick_action:
hoReadyToRecieve_ToLeft := FALSE;
END_ACTION

ACTION WaitToPlace_action:
hoPartAvail_ToRight := TRUE;
END_ACTION

ACTION Place_entry:
bPlace   := TRUE;
bPicked := FALSE;
END_ACTION

ACTION Place_action:
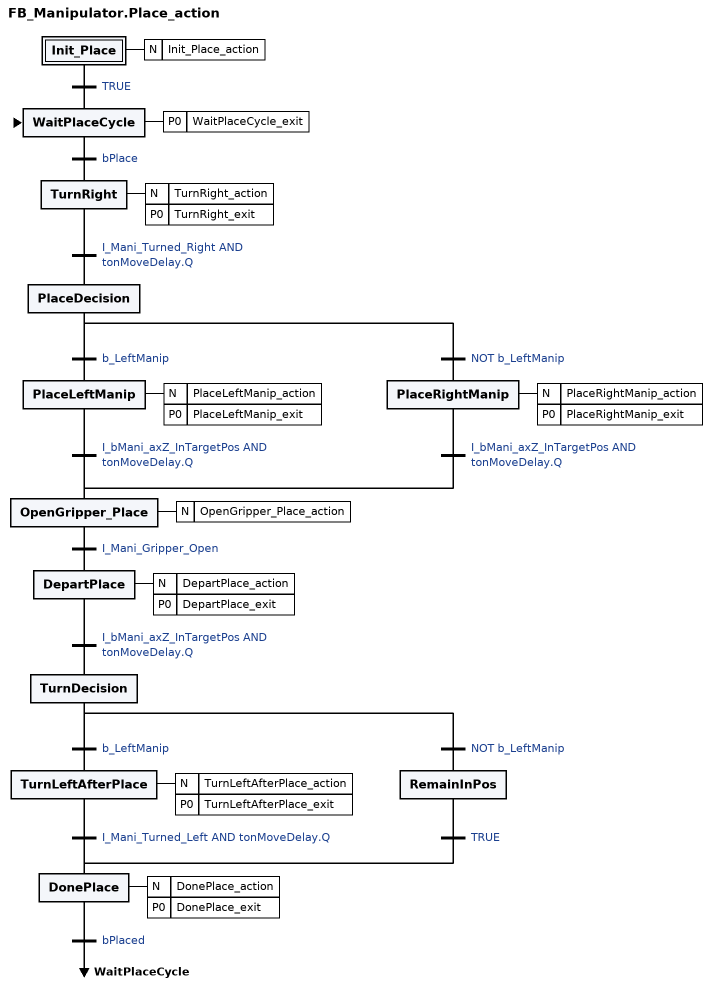
INITIAL_STEP Init_Place:
	Init_Place_action(N);
END_STEP
TRANSITION FROM Init_Place TO WaitPlaceCycle := TRUE;
END_TRANSITION
STEP WaitPlaceCycle:
	WaitPlaceCycle_exit(P0);
END_STEP
TRANSITION FROM WaitPlaceCycle TO TurnRight := bPlace;
END_TRANSITION
STEP TurnRight:
	TurnRight_action(N);
	TurnRight_exit(P0);
END_STEP
TRANSITION FROM TurnRight TO PlaceDecision := I_Mani_Turned_Right AND tonMoveDelay.Q;
END_TRANSITION
STEP PlaceDecision:
END_STEP
TRANSITION FROM PlaceDecision TO PlaceLeftManip := b_LeftManip;
END_TRANSITION
TRANSITION FROM PlaceDecision TO PlaceRightManip := NOT b_LeftManip;
END_TRANSITION
STEP PlaceLeftManip:
	PlaceLeftManip_action(N);
	PlaceLeftManip_exit(P0);
END_STEP
TRANSITION FROM PlaceLeftManip TO OpenGripper_Place := I_bMani_axZ_InTargetPos AND tonMoveDelay.Q;
END_TRANSITION
STEP PlaceRightManip:
	PlaceRightManip_action(N);
	PlaceRightManip_exit(P0);
END_STEP
TRANSITION FROM PlaceRightManip TO OpenGripper_Place := I_bMani_axZ_InTargetPos AND tonMoveDelay.Q;
END_TRANSITION
STEP OpenGripper_Place:
	OpenGripper_Place_action(N);
END_STEP
TRANSITION FROM OpenGripper_Place TO DepartPlace := I_Mani_Gripper_Open;
END_TRANSITION
STEP DepartPlace:
	DepartPlace_action(N);
	DepartPlace_exit(P0);
END_STEP
TRANSITION FROM DepartPlace TO TurnDecision := I_bMani_axZ_InTargetPos AND tonMoveDelay.Q;
END_TRANSITION
STEP TurnDecision:
END_STEP
TRANSITION FROM TurnDecision TO TurnLeftAfterPlace := b_LeftManip;
END_TRANSITION
TRANSITION FROM TurnDecision TO RemainInPos := NOT b_LeftManip;
END_TRANSITION
STEP TurnLeftAfterPlace:
	TurnLeftAfterPlace_action(N);
	TurnLeftAfterPlace_exit(P0);
END_STEP
TRANSITION FROM TurnLeftAfterPlace TO DonePlace := I_Mani_Turned_Left AND tonMoveDelay.Q;
END_TRANSITION
STEP RemainInPos:
END_STEP
TRANSITION FROM RemainInPos TO DonePlace := TRUE;
END_TRANSITION
STEP DonePlace:
	DonePlace_action(N);
	DonePlace_exit(P0);
END_STEP
TRANSITION FROM DonePlace TO WaitPlaceCycle := bPlaced;
END_TRANSITION

ACTION Init_Place_action:
bPlaced := FALSE;
END_ACTION

ACTION WaitPlaceCycle_exit:
bPlaced := FALSE;
END_ACTION

ACTION TurnRight_action:
tonMoveDelay(IN:=TRUE , PT:= tMoveDelay);
O_Mani_Turn_Right	 := TRUE;
O_Mani_Turn_Left 	 := FALSE;
END_ACTION

ACTION TurnRight_exit:
tonMoveDelay(IN:=FALSE);
END_ACTION

ACTION PlaceLeftManip_action:
tonMoveDelay(IN:=TRUE , PT:= tMoveDelay);
O_fMani_axZ_Velo :=10;
O_fMani_axZ_TargetPos := -74;
O_bMani_axZ_Start := TRUE;
END_ACTION

ACTION PlaceLeftManip_exit:
O_bMani_axZ_Start 	:= FALSE;
tonMoveDelay(IN		:=FALSE);
END_ACTION

ACTION PlaceRightManip_action:
tonMoveDelay(IN:=TRUE , PT:= tMoveDelay);
O_fMani_axZ_Velo :=10;
O_fMani_axZ_TargetPos := -120;
O_bMani_axZ_Start := TRUE;
END_ACTION

ACTION PlaceRightManip_exit:
O_bMani_axZ_Start := FALSE;
tonMoveDelay(IN:=FALSE);
END_ACTION

ACTION OpenGripper_Place_action:
O_Mani_Gripper_Close := FALSE;
END_ACTION

ACTION DepartPlace_action:
tonMoveDelay(IN:=TRUE , PT:= tMoveDelay);
O_fMani_axZ_Velo :=10;
O_fMani_axZ_TargetPos := -40;
O_bMani_axZ_Start := TRUE;
END_ACTION

ACTION DepartPlace_exit:
O_bMani_axZ_Start := FALSE;
tonMoveDelay(IN:=FALSE);
END_ACTION

ACTION TurnLeftAfterPlace_action:
tonMoveDelay(IN:=TRUE , PT:= tMoveDelay);
O_Mani_Turn_Right	 := FALSE;
O_Mani_Turn_Left 	 := TRUE;
END_ACTION

ACTION TurnLeftAfterPlace_exit:
tonMoveDelay(IN:=FALSE);
END_ACTION

ACTION DonePlace_action:
bPlaced				:= TRUE;
END_ACTION

ACTION DonePlace_exit:
bPlaced := FALSE;
END_ACTION
END_ACTION

ACTION Place_exit:
bPlace := FALSE;
bPicked := FALSE;
END_ACTION

ACTION Handshake_Place_action:
hoPartAvail_ToRight := FALSE;
END_ACTION

ACTION SFCResetStep_action:
SFCReset := TRUE;
END_ACTION
END_FUNCTION_BLOCK

(* POU PRG/PRG_ManipulatorRight, ST *)
PROGRAM PRG_ManipulatorRight
VAR_INPUT
	(* PackML Inputs *)
	State							: E_PackMLState;
	ControlMode					: E_Mode;
	ProceeduralMode				: E_ModeProc;

	hiPartAvail_FromLeft			: BOOL;
	hiRdyToReceive_FromRight  : BOOL;
END_VAR
VAR_OUTPUT
	(* PackML Outputs *)
	SC								: BOOL;
	bInitDone						: BOOL;
	bStopOk						: BOOL;

	hoReadyToRecieve_ToLeft	: BOOL;
	hoPartAvail_ToRight			: BOOL;
END_VAR
VAR
	initOK							: BOOL := FALSE;
	fbManipulatorRight 				: FB_Manipulator;
	fbManipulatorLeft: BOOL;
END_VAR
SC := FALSE;

CASE State OF
	eSt_Aborting:
		O_ManiL_Turn_Left		 		:= FALSE;
		O_ManiL_Turn_Right		 		:= FALSE;
		bManiL_axZ_Start					:= FALSE;
		IF I_ManiL_Gripper_Open THEN
			O_ManiL_Gripper_Close 	:= FALSE;
		ELSE
			O_ManiL_Gripper_Close		:= TRUE;
		END_IF
		SC := TRUE;
	eSt_Clearing:
		SC := TRUE;
	;
	eSt_Resetting:
		SC := TRUE
	;

	eSt_Starting:
		IF NOT  fbManipulatorRight.bInitialised THEN
			actUpdateIO;
		ELSE
			bInitDone	 := TRUE;
			SC		 	 := TRUE;
		END_IF
	;
	eSt_Holding:
	;
	eSt_UnHolding:
	;
	eSt_Suspending:
		fbManipulatorRight (I_Enable :=  FALSE);
		actUpdateIO;
		IF fbManipulatorRight.bStopOk THEN
			SC := TRUE;
		END_IF
	eSt_Unsuspending:
		SC := TRUE;
	eSt_Execute:
		CASE ControlMode OF
			eMode_Automatic:
				fbManipulatorRight (
					I_Enable						:=  TRUE,
					I_Reset						:=   ,);
				actUpdateIO;
			eMode_Manual:
			;
		END_CASE
		eSt_Completing:
		;
	
		eSt_Stopping:
			fbManipulatorRight (I_Enable :=  FALSE);
			actUpdateIO;
			IF fbManipulatorRight.bStopOk THEN
				bStopOk := TRUE;
				SC 	   := TRUE;
			ELSE
				bStopOk := FALSE;
			END_IF
END_CASE
END_PROGRAM
ACTION actUpdateIO:
fbManipulatorRight (
					b_LeftManip					:= FALSE ,
					I_Mani_Limit_Up				:= I_ManiR_Limit_Up,
					I_Mani_Limit_Dn				:= I_ManiR_Limit_Dn,
					I_Mani_Limit_Home			:= I_ManiR_Limit_Home ,
					I_Mani_Turned_Left			:= I_ManiR_Turned_Left,
					I_Mani_Turned_Right			:= I_ManiR_Turned_Right ,
					I_Mani_Gripper_Open		:= I_ManiR_Gripper_Open ,
					I_fMani_axZ_CurrPos			:= fManiR_axZ_CurrPos ,
					I_bMani_axZ_InTargetPos	:= bManiR_axZ_InTargetPos,

					hiPartAvail_FromLeft			:= hiPartAvail_FromLeft ,
					hiRdyToReceive_FromRight	:= hiRdyToReceive_FromRight,
					hoReadyToRecieve_ToLeft	=> hoReadyToRecieve_ToLeft,
					hoPartAvail_ToRight			=> hoPartAvail_ToRight ,
			
					O_Mani_Turn_Left			=> O_ManiR_Turn_Left ,
					O_Mani_Turn_Right			=> O_ManiR_Turn_Right ,
					O_Mani_Gripper_Close		=> O_ManiR_Gripper_Close ,
					O_bMani_axZ_Enable		=> bManiR_axZ_Enable ,
					O_bMani_axZ_Start			=> bManiR_axZ_Start ,
					O_fMani_axZ_Velo			=> fManiR_axZ_Velo,
					O_fMani_axZ_TargetPos		=> fManiR_axZ_TargetPos );
END_ACTION

(* POU Examples/PRG_MAIN_SAMPLE, ST *)
PROGRAM PRG_MAIN_SAMPLE
VAR
	fbStateModel		: FB_PackMLStateModel_ST;	(*FB for executing PackML state model*)
	bBlink				: BOOL;	(*1s blinkg for CodeSys Simulation*)
	c					: INT;	(*Support variable for blinking*)
END_VAR
(* ****** Section 1: Initialisations and default values. Initial conditions for variables on every PLC cycle*)
fbStateModel.bSC := FALSE;

(* ****** Section 2: Actions in your program without considering the Control Mode. I.e. actions are performed same way indenpendent on
current Control Mode selection.*)
(*Mode independent state actions*)
CASE fbStateModel.eState OF
eSt_Aborting:
	(* One can make specific actions in case of specific Mode-State combination.
	   One can also consider to call a specific program when in specific Mode-State combination*)
	actAborting;
	fbStateModel.bSC := TRUE;		(*TODO: Remove/Replace this row with desired actions*)
eSt_Clearing:
	fbStateModel.bSC := TRUE;		(*TODO: Remove/Replace this row with desired actions*)
eSt_Stopping:
	fbStateModel.bSC := TRUE;		(*TODO: Remove/Replace this row with desired actions*)
eSt_Resetting:
	fbStateModel.bSC := TRUE;		(*TODO: Remove/Replace this row with desired actions*)
eSt_Holding:
	fbStateModel.bSC := TRUE;		(*TODO: Remove/Replace this row with desired actions*)
eSt_UnHolding:
	fbStateModel.bSC := TRUE;		(*TODO: Remove/Replace this row with desired actions*)
eSt_Suspending:
	fbStateModel.bSC := TRUE;		(*TODO: Remove/Replace this row with desired actions*)
eSt_Unsuspending:
	fbStateModel.bSC := TRUE;		(*TODO: Remove/Replace this row with desired actions*)
END_CASE;

(* ****** Section 3: Actions in your program which are Control Mode specific. Two nested case structures where outer one selects the
control mode and inner the PackML state. In order to avoid conflicts, it would be better to process each PackML state either in Section 2 
or Section 3, but not in both. *)
(*Execution mode related state actions*)
CASE fbStateModel.eMode OF
(*MODE: MANUAL*)
eMode_Manual:
	(* ****** Section 3.1: PackML state based processing actions when Control Mode is Manual.*)
	CASE fbStateModel.eState OF
	eSt_Idle:
		fbStateModel.bAck_Completed := FALSE;		(*TODO: Remove/Replace this row with desired actions*)
	eSt_Starting:
		fbStateModel.bSC := TRUE;					(*TODO: Remove/Replace this row with desired actions*)
	eSt_Completing:
		fbStateModel.bSC := TRUE;					(*TODO: Remove/Replace this row with desired actions*)
	eSt_Completed:
		fbStateModel.bAck_Completed := TRUE;		(*TODO: Remove/Replace this row with desired actions*)
	END_CASE;

(*MODE: AUTOMATIC*)
eMode_Automatic:
	(* ****** Section 3.2: PackML state based processing actions when Control Mode is Automatic.*)
	CASE fbStateModel.eState OF
	eSt_Idle:
		fbStateModel.bAck_Completed := FALSE;		(*TODO: Remove/Replace this row with desired actions*)
	eSt_Starting:
		fbStateModel.bSC := TRUE;					(*TODO: Remove/Replace this row with desired actions*)
	eSt_Completing:
		fbStateModel.bSC := TRUE;					(*TODO: Remove/Replace this row with desired actions*)
	eSt_Completed:
		;
		(*fbStateModel.bAck_Completed:= I_Btn_Start;*)
	END_CASE;

(*MODE: UNKNOWN*)
ELSE	(*This is an Error branch.*)
	; (*TODO: Make implementation*)
END_CASE;

(* ****** Section 4: Grouping PackML states for calling Programs or FB instances.
This is to avoid repetition inside case structure in Section 3. With IF clause setting lower (and upper) state limits we can filter out the states when we want to call 
specific programs. The order of states is defined in Tab:Data types > E_PackMLState. eSt_Aborting is lowest and eSt_Completed is highest.
Here we filter calling programs, only when we are in higher states than Stopped. Inside IF there is again CASE which process each Control Mode separately.*)
(*Execution part. Making calls for program if we are on states above Stopped*)
IF (fbStateModel.eState > eSt_Stopped) THEN
	CASE fbStateModel.eMode OF
		(*MODE: MANUAL*)
		eMode_Manual:
			;
		(*MODE: AUTOMATIC*)
		eMode_Automatic:
			;
	END_CASE;
END_IF;

(* ****** Section 5: Calling the fbStateModel instance.
Here the instance of state model is called and all triggering inputs are set, but bSC (State Completed), which you control in your programs. 
This is indication that your program has  finished certain stage.
- Pay attention where the instance fbStateModel is defined. Do you do it in global variables or e.g. here in PRG_MAIN? Important is to use the 
same instance in all places, so that machine state is unique and shared. Remember, if you have multiple definitions, the PRG_MAIN "hides" 
the global one, and might lead to problems elswhere, when you think you are using the same instance, but actually are not. 
- In case you are using the PackML visualisation (VC_PackMLStates), make sure you connect its placeholder to the very same PackML FB instance.
- The Mask for wIgnoreState is created as following. I use binary base for the value(2#). The lowest bit in the mask corresponds the eSt_Aborting
 in E_PackMLState. The next is eSt_Aborted, and so on. Specific state is ignored and jumped over when it is masked out i.e. ignored by having 1 
in that position. Note that implementation allows this only for selected states. See FB_PackMLStateModel_ST code for further details.*)
(*Calling & Updating the state model*)
(*TODO: Evaluate and change all input conditions according your application needs*)
fbStateModel(
	bResetFB:= ,
	eModeReq:= ,
	wIgnoreState := 2#000000,		(*TODO: Which states should be ignodered. Default: 2#000000 or 2#100000*)
	bSC:= ,		(*Must NOT be assigned ANY variable, because fb input is directly assigned above by your programs!!!*)
	bAbort:= ,
	bClear:= ,
	bReset:= ,
	bStart:= ,
	bHold:= ,
	bUn_Hold:= ,
	bSuspend:= ,
	bUn_Suspend:= ,
	bStop:= ,
	bComplete:= ,
	bAck_Completed:= ,
	eMode=> ,
	eState=> );

(* ****** Section 6: Here we update all outputs according the current state of our PackML model. This allows us to process the in single location.
The control of outputs is bind to state, not e.g. to inputs. The inputs are the one driving the PackML model forward. Again CASE structure can be used.*)
(*Call for HMI and UI update*)
HMI_and_UI_Update;
END_PROGRAM
ACTION actAborting:
(*You can add here Aborting related actions as one central collection.
This action can be called from multiple places, in case needed, 
but is part of program*)
;
END_ACTION
ACTION HMI_and_UI_Update:
(*HMI Update*)
(*Calling blinking sub-program*)
(*PRG_Blinking (bSign4Hz=> , bSign2Hz=> , bSign1Hz=> , bSign0_5Hz=> );*)
(*Codesys simulation 1Hz blinking*)
c:= c + 1;
IF c > 1 THEN
	c:=0;
END_IF;
bBlink := (c=0);	(*bBlink is true if c=0*)

(*Init values*)
O_Light_Stop := FALSE;	(*TODO: Change initial values according your app needs*)

(*TODO: Change values according range of states *)
(*Start light*)
(*O_Light_Start :=  (fbStateModel.eState >= eSt_Resetting) AND (fbStateModel.eState < eSt_Completed); *)

(*TODO: Change output values according states *)
CASE fbStateModel.eState OF
eSt_Aborting, eSt_Aborted:
	O_Light_Stop := bBlink;					(*TODO: Change initial values according your app needs*)
eSt_Clearing:
	O_Light_Stop := bBlink; 					(*TODO: Change initial values according your app needs*)
eSt_Stopping, eSt_Stopped, eSt_Completed:
	O_Light_Stop := TRUE;					(*TODO: Change initial values according your app needs*)
eSt_Starting:
	;
	(*O_Light_Start := bBlink;	*)				(*TODO: Change initial values according your app needs*)
END_CASE;
END_ACTION

(* POU FBs/FB_PackMLStateModel_ST, ST *)
FUNCTION_BLOCK FB_PackMLStateModel_ST
(*PackML State model implementation for applications.
Author: Niko Siltala, niko.siltala@tut.fi, Tampere University of Technology / MEI
Date: 2016-12-12
Version: 1.0
*)
VAR_INPUT
	bResetFB	: BOOL;		(*Resets whole FB*)
	eModeReq	: E_Mode;	(*Requested mode*)
	wIgnoreState: DWORD;	(*Ignoring states. See bit from E_PackMLState definition. Aborting = bit0*)
	bSC			: BOOL;		(*Step Completed acknoledgement*)
	bAbort		: BOOL;		(*Abortting signal = EmergencyStop*)
	bClear		: BOOL;		(*Clear signal*)
	bReset		: BOOL;		(*Reseting signal*)
	bStart		: BOOL;		(*Start signal*)
	bHold		: BOOL;		(*Hold signal*)
	bUn_Hold	: BOOL;		(*Un-Hold signal*)
	bSuspend	: BOOL;		(*Suspend signal*)
	bUn_Suspend	: BOOL;		(*Un-Suspend signal*)
	bStop		: BOOL;		(*Stop signal*)
	bComplete	: BOOL;		(*Complete signal*)
	bAck_Completed	: BOOL;	(*Acknoledgement for Complete signal*)
END_VAR
VAR_OUTPUT
	eMode	: E_Mode;		(*Current mode*)
	eState	: E_PackMLState;(*Current state*)
	strState : STRING(15);		(*State as String*)
END_VAR
VAR
	RTrig_bSC		: R_TRIG; 		(*Rising trigger for State Completed*)
	RTrig_StateChange : R_TRIG; 	(*Rising trigger for State signal*)
	bResetLocal		: BOOL:=FALSE;	(*Paikallinen Reset*)
	bInitDone		: BOOL;			(*Initialisation*)
END_VAR
IF bResetFB THEN	(*Reseting FB*)
	bInitDone := FALSE;
END_IF;

(*Initialisation*)
IF NOT bInitDone THEN
	eState:= eSt_Aborting;
	strState:='Aborting';
	bInitDone:=TRUE;
END_IF;

(*Rising triggers monitor*)
RTrig_bSC(CLK:=bSC , Q=> );

(*Abort signal interrupt*)
IF bAbort AND (eState > eSt_Clearing) THEN
	eState:=eSt_Aborting;
END_IF;

(*Stop signal interrupt*)
IF bStop AND (eState > eSt_Stopping) THEN
	eState:=eSt_Stopping;
END_IF;


(*Main case structure*)
CASE eState OF
eSt_Aborting:
	strState:='Aborting';
	IF bSC THEN
		eState:=eSt_Aborted;
	END_IF;

eSt_Aborted:
	strState:='Aborted';
	eMode:=eModeReq;	(*Change Mode allowed*)
	IF bClear AND NOT bAbort THEN
		eState:=eSt_Clearing;
	END_IF;

eSt_Clearing:
	strState:='Clearing';
	IF bAbort THEN
		eState:=eSt_Aborting;
	ELSIF bSC THEN
		eState:=eSt_Stopped;
		RTrig_StateChange(CLK:=bReset , Q=> );
	END_IF;

eSt_Stopping:
	strState:='Stopping';
	IF bSC THEN
		eState:=eSt_Stopped;
		RTrig_StateChange(CLK:=bReset , Q=> );
	END_IF;

eSt_Stopped:
	strState:='Stopped';
	eMode:=eModeReq;	(*Change Mode allowed*)
	RTrig_StateChange(CLK:=bReset , Q=> );
(*	ELSIF NOT bStop AND (RTrig_StateChange.Q OR (wIgnoreState.5 AND bStart) ) THEN*)
	IF NOT bStop THEN	(*Stop signal is not active.*)
		IF wIgnoreState.5 AND bStart THEN	(*Reset state is ignored and going directly to start *)
			eState:=eSt_Idle;
(*		ELSIF RTrig_StateChange.Q THEN 	(*Rising edge for reset*)*)
		ELSIF bReset THEN 	(*Reset*)
			eState:=eSt_Resetting;
		END_IF;
	END_IF;

eSt_Resetting:
	strState:='Resetting';
	IF bSC OR wIgnoreState.5 THEN
		eState:=eSt_Idle;
	END_IF;

eSt_Idle:
	strState:='Idle';
	eMode:=eModeReq;	(*Change Mode allowed*)
	IF bStart OR wIgnoreState.6 THEN (* IDLE state is ignoered*)
		eState:=eSt_Starting;
	END_IF;

eSt_Starting:
	strState:='Starting';
	IF bSC OR wIgnoreState.7 THEN (* STARTING state is ignoered*)
		eState:=eSt_Execute;
	END_IF;

eSt_Execute:
	strState:='Execute';
	IF bComplete THEN
		eState:=eSt_Completing;
	ELSIF bHold THEN
		eState:=eSt_Holding;
	ELSIF bSuspend THEN
		eState:=eSt_Suspending;
	END_IF;

eSt_Holding:
	strState:='Holding';
	IF bSC THEN
		eState:=eSt_Held;
	END_IF;

eSt_Held:
	strState:='Held';
	IF bUn_Hold AND NOT bHold THEN
		eState:=eSt_UnHolding;
	END_IF;

eSt_UnHolding:
	strState:='Un-Holding';
	IF bSC THEN
		eState:=eSt_Execute;
	END_IF;

eSt_Suspending:
	strState:='Suspending';
	IF bSC THEN
		eState:=eSt_Suspended;
	END_IF;

eSt_Suspended:
	strState:='Suspended';
	IF bUn_Suspend AND NOT bSuspend THEN
		eState:=eSt_Unsuspending;
	END_IF;

eSt_Unsuspending:
	strState:='Un-Suspending';
	IF bSC THEN
		eState:=eSt_Execute;
	END_IF;

eSt_Completing:
	strState:='Completing';
	IF RTrig_bSC.Q THEN
		eState:=eSt_Completed;
	END_IF;

eSt_Completed:
	strState:='Completed';
	IF bReset OR bAck_Completed THEN
		eState:=eSt_Resetting;
	END_IF;

ELSE
	(*Default error handler. Undefined state set*)
	eState:=eSt_Aborting;
END_CASE;
END_FUNCTION_BLOCK

(* POU Examples/Processes/PRG_ProcessAuto, SFC *)
PROGRAM PRG_ProcessAuto
VAR_INPUT
	bReset	: BOOL;	(*Reset program*)
	bEnable	: BOOL;	(*enable and run*)
END_VAR
VAR
	tonDelay		: TON;
	SFCReset		: BOOL;
END_VAR
VAR CONSTANT
	tDelayTime		: TIME := t#2s;	(*Delay time for timer*)
END_VAR
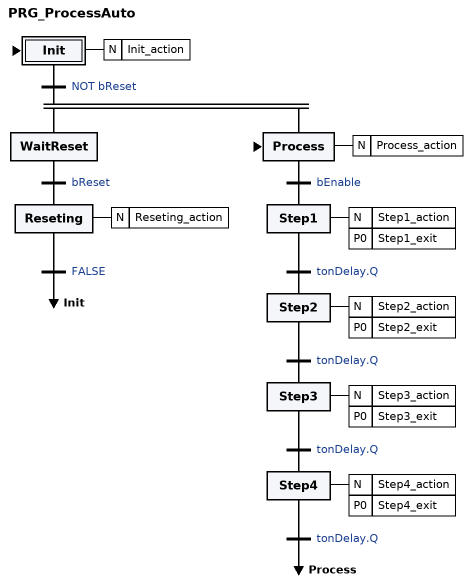
INITIAL_STEP Init:
	Init_action(N);
END_STEP
TRANSITION FROM Init TO (WaitReset, Process) := NOT bReset;
END_TRANSITION
STEP WaitReset:
END_STEP
TRANSITION FROM WaitReset TO Reseting := bReset;
END_TRANSITION
STEP Process:
	Process_action(N);
END_STEP
TRANSITION FROM Process TO Step1 := bEnable;
END_TRANSITION
STEP Step1:
	Step1_action(N);
	Step1_exit(P0);
END_STEP
TRANSITION FROM Step1 TO Step2 := tonDelay.Q;
END_TRANSITION
STEP Step2:
	Step2_action(N);
	Step2_exit(P0);
END_STEP
TRANSITION FROM Step2 TO Step3 := tonDelay.Q;
END_TRANSITION
STEP Step3:
	Step3_action(N);
	Step3_exit(P0);
END_STEP
TRANSITION FROM Step3 TO Step4 := tonDelay.Q;
END_TRANSITION
STEP Step4:
	Step4_action(N);
	Step4_exit(P0);
END_STEP
TRANSITION FROM Step4 TO Process := tonDelay.Q;
END_TRANSITION
STEP Reseting:
	Reseting_action(N);
END_STEP
TRANSITION FROM Reseting TO Init := FALSE;
END_TRANSITION

ACTION Init_action:
SFCReset := FALSE;
END_ACTION

ACTION Process_action:
O_Light_1 :=FALSE;
O_Light_2 :=FALSE;
O_Light_3 :=FALSE;
O_Light_4 :=FALSE;

tonDelay(IN:=FALSE , PT:=tDelayTime);
END_ACTION

ACTION Step1_action:
O_Light_1 := TRUE;

tonDelay(IN:=TRUE);
END_ACTION

ACTION Step1_exit:
tonDelay(IN:=FALSE);
END_ACTION

ACTION Step2_action:
O_Light_2 := TRUE;

tonDelay(IN:=TRUE);
END_ACTION

ACTION Step2_exit:
tonDelay(IN:=FALSE);
END_ACTION

ACTION Step3_action:
O_Light_3 := TRUE;

tonDelay(IN:=TRUE);
END_ACTION

ACTION Step3_exit:
tonDelay(IN:=FALSE);
END_ACTION

ACTION Step4_action:
O_Light_4 := TRUE;

tonDelay(IN:=TRUE);
END_ACTION

ACTION Step4_exit:
tonDelay(IN:=FALSE);
END_ACTION

ACTION Reseting_action:
SFCReset := TRUE;
END_ACTION
END_PROGRAM

(* POU Examples/Processes/PRG_ProcessManual, ST *)
PROGRAM PRG_ProcessManual
VAR_INPUT
	bReset	: BOOL;	(*Reset program*)
	bNext	: BOOL;	(*Next step*)
END_VAR
VAR
	iStep	: INT;	(*Step variable*)
	rtTrigger	: R_TRIG;	(*Trigger from button*)
END_VAR
rtTrigger(CLK:=bNext , Q=> );
IF  rtTrigger.Q THEN
	iStep := iStep + 1;
	IF iStep >= 5 THEN
		iStep := 1;
	END_IF
END_IF;

(*Default values*)
	O_Light_1 := FALSE;
	O_Light_2 := FALSE;
	O_Light_3 := FALSE;
	O_Light_4 := FALSE;

CASE iStep OF
0:
	;
1:
	O_Light_1 := TRUE;
2:
	O_Light_2 := TRUE;
3:
	O_Light_3 := TRUE;
4:
	O_Light_4 := TRUE;
ELSE
	iStep := 0;
END_CASE
END_PROGRAM

(* POU Examples/PRG_SFC_Example, SFC *)
PROGRAM PRG_SFC_Example
VAR_INPUT
	bReset		: BOOL;	(*Reset Request*)
END_VAR
VAR_OUTPUT
END_VAR
VAR
	bLocalReset	: BOOL;	(*Performs local reset*)
	SFCReset 	: BOOL;	(*Resets the execution of SFC to init once this SFCFlag is set true *)
END_VAR
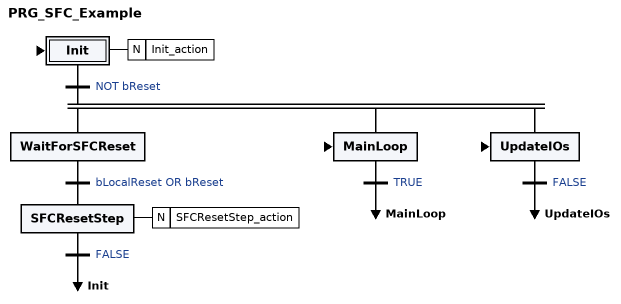
INITIAL_STEP Init:
	Init_action(N);
END_STEP
TRANSITION FROM Init TO (WaitForSFCReset, MainLoop, UpdateIOs) := NOT bReset;
END_TRANSITION
STEP WaitForSFCReset:
END_STEP
TRANSITION FROM WaitForSFCReset TO SFCResetStep := bLocalReset OR bReset;
END_TRANSITION
STEP SFCResetStep:
	SFCResetStep_action(N);
END_STEP
TRANSITION FROM SFCResetStep TO Init := FALSE;
END_TRANSITION
STEP MainLoop:
END_STEP
TRANSITION FROM MainLoop TO MainLoop := TRUE;
END_TRANSITION
STEP UpdateIOs:
END_STEP
TRANSITION FROM UpdateIOs TO UpdateIOs := FALSE;
END_TRANSITION

ACTION Init_action:
SFCReset := FALSE;
bLocalReset	:= FALSE;
END_ACTION

ACTION SFCResetStep_action:
SFCReset := TRUE;
END_ACTION
END_PROGRAM

(* POU Simulation/PRG_Simulator, ST *)
PROGRAM PRG_Simulator
(*This Program is simulating the real machine and mimics its behaviour.
The main task is to update the inputs for students program according the stimulus student provides as outputs.
Another task is to monitor (physical) error conditions occuring in the system and record them.
Author: Niko Siltala, niko.siltala@tut.fi, Tampere University of Technology / MEI
Date: 2016-12-12
Version: 1.0
*) 
VAR
	bBtn_EmergencyStop	: BOOL;	(*Emergency Stop button*)
	rsEmergencyClear	: RS;	(*RS - flip-flop for Emergency clear info*)
	i 	: INT;
	c 	: INT;
	fbManipLeft		: FB_Simu_Manipulator;	(*Left simulated manipulator *)
	fbManipRight	: FB_Simu_Manipulator;	(*Right simulated manipulator *)
	fbDrill			: FB_Simu_Drill;		(*Drill machine simulated*)
	arrParts_ConvIn		: ARRAY [0..10] OF ST_Part; (*Parts on input conveyour*)
	arrParts_ConvOut	: ARRAY [0..10] OF ST_Part; (*Parts on output conveyour*)
	stPart_inMLeftGripper 	: ST_Part; 	(*Data structure for the part*)
	stPart_inMRightGripper 	: ST_Part; 	(*Data structure for the part*)
	stPart_inDrillFixture 	: ST_Part; 	(*Data structure for the part*)
	bAddPartOnConvIn	: BOOL;	(*Adds new part on conveyor*)
	bClearErrors		: BOOL;	(*Clear Errors*)
	bClearSystem		: BOOL;	(*Clears system from parts *)
	RT_AddPart			: R_TRIG;
	wError_ManipL			: WORD;	(*Error bits between convIn and Manip_Left*)
	wError_Drill		: WORD; (*Error bits at drill*)
	wError_ManipR		: WORD;	(*Error bits between convIn and Manip_Left*)
	iState_IF			: ARRAY [1..5] OF UINT;	(*State variable; Exchange between 1=ConvIn->ManipL, 2=ManipL->Drill, 3=Drill->ManipR, 4=ManipR->ConvOut, 5=Drill*)
	tofPartLeavesConvOut	: TOF;	(*Off timer for out sensor*)
END_VAR
VAR CONSTANT
	bMANUAL_CONTROLS				: BOOL 	:=FALSE;(*Manual override for controls*)
	fPOS_MANIP_CONV_NO_PART_SAFE	: REAL	:= 90;	(*Manipulator on conv with NO part - Safe to move*)
	fPOS_MANIP_CONV_WITH_PART_SAFE	: REAL	:= 70;	(*Manipulator on conv with part - Safe to move*)
	fPOS_MANIP_CONV_PICK_LEVEL		: REAL	:= 120;	(*Manipulator Pick/place level on conv*)
	fPOS_MANIP_DRILL_WITH_PART_SAFE	: REAL	:= 53;	(*Manipulator coming to drill with part - Safe to move*)
	fPOS_MANIP_DRILL_NO_PART_SAFE	: REAL	:= 46;	(*Manipulator coming to drill with NO part - Safe to move*)
	fPOS_MANIP_DRILL_PICK_LEVEL		: REAL	:= 74;	(*Manipulator Pick/place level on Drill*)
	fPOS_MANIP_PICK_TOLERANCE		: REAL	:= 30;	(*Manipulator Pick level tolerance from the part (=fingers length)*)
	fPART_HEIGH						: REAL	:= 50;	(*Part height*)
	fPART_PICK_TOLERANCE			: REAL	:= 10;	(*Part pick & place (negative) tolerance from Levels.*)
	fPART_HOLE_DEPTH_REQ			: REAL	:= 40;	(*Part required Hole depth*)
	fPART_HOLE_DEPTH_MAX			: REAL	:= 45;	(*Max Hole depth*)
	fPOS_DRILL_BIT_TOUCHES			: REAL	:= 100;	(*Drill touches the part*)
	iDRILL_SPINDLE_MIN_FOR_DRILLING	: INT	:= 400;	(*Minimum spindle speed for drilling*)
END_VAR
(*Handle counter*)
c:= c+1;
IF c> 10 THEN
	c:= 0;
END_IF;

(*Simulate emergency stop circuitry*)
rsEmergencyClear(
	SET:= I_Btn_Reset,
	RESET1:= bBtn_EmergencyStop,
	Q1=> I_EmergencyClear);

(*Adds new parts on input conveyour*)
RT_AddPart(CLK:=bAddPartOnConvIn , Q=> );
IF RT_AddPart.Q AND NOT arrParts_ConvIn[5].bExists THEN
	arrParts_ConvIn[5].bExists := TRUE;
END_IF;

(*Input Conveyour Simulation*)
IF O_ConvIn_MotON THEN
	IF (c MOD 5) = 0 THEN
		(*Move parts forward*)
		F_MovePartForward(arrParts_ConvIn);
	END_IF;
END_IF;
(*Part in pick postition*)
I_ConvIn_PartPresent := arrParts_ConvIn[0].bExists;

(*Output Conveyour Simulation*)
IF O_ConvOut_MotON THEN
	IF (c MOD 5) = 0 THEN
		(*Move parts forward*)
		F_MovePartForward(arrParts_ConvOut);
	END_IF;
END_IF;
(*Part in end postition*)
I_ConvOut_PartPresent := arrParts_ConvOut[0].bExists;
tofPartLeavesConvOut(
	IN:=arrParts_ConvOut[0].bExists ,
	PT:= T#1s,
	Q=>I_ConvOut_PartPresent );
IF arrParts_ConvOut[0].bExists THEN
	(*Clear part at end of output conveyour*)
	arrParts_ConvOut[0].bExists := FALSE;
	arrParts_ConvOut[0].bHasHole := FALSE;
END_IF;


IF bMANUAL_CONTROLS THEN
	(*Left manipulator*)
	fbManipLeft(
		bEnable:= ,
		bLift_Start:= ,
		fLift_Velo:= ,
		fLift_TargetPos:= ,
		bBeam_Left:= ,
		bBeam_Right:= ,
		bGripper_Close:= ,
		stPart_inGripper:= stPart_inMLeftGripper,
		bGripperIsOpen=> I_ManiL_Gripper_Open,
		bLift_InTarget=> bManiL_axZ_InTargetPos,
		fLift_CurrentPos=> fManiL_axZ_CurrPos,
		bLimit_Top=> I_ManiL_Limit_Up,
		bLimit_Bottom=> I_ManiL_Limit_Dn,
		bHome_Sensor=> I_ManiL_Limit_Home,
		bBeamAtRight=> I_ManiL_Turned_Right,
		bBeamAtLeft=> I_ManiL_Turned_Left);
	
	(*Right manipulator*)
	fbManipRight(
		bEnable:= ,
		bLift_Start:= ,
		fLift_Velo:= , 
		fLift_TargetPos:= , 
		bBeam_Left:= ,
		bBeam_Right:= ,
		bGripper_Close:= , 
		stPart_inGripper:= stPart_inMRightGripper,
		bGripperIsOpen=> I_ManiR_Gripper_Open,
		bLift_InTarget=> bManiR_axZ_InTargetPos,
		fLift_CurrentPos=> fManiR_axZ_CurrPos,
		bLimit_Top=> I_ManiR_Limit_Up,
		bLimit_Bottom=> I_ManiR_Limit_Dn,
		bHome_Sensor=> I_ManiR_Limit_Home,
		bBeamAtRight=> I_ManiR_Turned_Right,
		bBeamAtLeft=> I_ManiR_Turned_Left);
	
	(*Call drill machine*)
	fbDrill(
		bEnable:= ,
		bLift_Start:= ,
		fLift_Velo:= ,
		fLift_TargetPos:= , 
		bDrillOn:= , 
		bFixture_Close:= , 
		stPart_inFixture:= stPart_inDrillFixture,
		bLift_InTarget=> bDrill_axZ_InTargetPos,
		fLift_CurrentPos=> fDrill_axZ_CurrPos,
		bLimit_Top=> I_Drill_Limit_Up,
		bLimit_Bottom=> I_Drill_Limit_Dn,
		bHome_Sensor=> I_Drill_Limit_Home,
		bFixture_Open=> I_Drill_Fixture_Open,
		bFixture_Closed=> I_Drill_Fixture_Closed);

ELSE
	(*Left manipulator*)
	fbManipLeft(
		bEnable:= bManiL_axZ_Enable,
		bLift_Start:= bManiL_axZ_Start,
		fLift_Velo:= fManiL_axZ_Velo,
		fLift_TargetPos:= fManiL_axZ_TargetPos,
		bBeam_Left:= O_ManiL_Turn_Left,
		bBeam_Right:= O_ManiL_Turn_Right,
		bGripper_Close:= O_ManiL_Gripper_Close,
		stPart_inGripper:= stPart_inMLeftGripper,
		bGripperIsOpen=> I_ManiL_Gripper_Open,
		bLift_InTarget=> bManiL_axZ_InTargetPos,
		fLift_CurrentPos=> fManiL_axZ_CurrPos,
		bLimit_Top=> I_ManiL_Limit_Up,
		bLimit_Bottom=> I_ManiL_Limit_Dn,
		bHome_Sensor=> I_ManiL_Limit_Home,
		bBeamAtRight=> I_ManiL_Turned_Right,
		bBeamAtLeft=> I_ManiL_Turned_Left);

	(*Right manipulator*)
	fbManipRight(
		bEnable:= bManiR_axZ_Enable,
		bLift_Start:= bManiR_axZ_Start,
		fLift_Velo:= fManiR_axZ_Velo,
		fLift_TargetPos:= fManiR_axZ_TargetPos,
		bBeam_Left:= O_ManiR_Turn_Left,
		bBeam_Right:= O_ManiR_Turn_Right,
		bGripper_Close:= O_ManiR_Gripper_Close,
		stPart_inGripper:= stPart_inMRightGripper,
		stPart_inGripper:= stPart_inMRightGripper,
		bGripperIsOpen=> I_ManiR_Gripper_Open,
		bLift_InTarget=> bManiR_axZ_InTargetPos,
		fLift_CurrentPos=> fManiR_axZ_CurrPos,
		bLimit_Top=> I_ManiR_Limit_Up,
		bLimit_Bottom=> I_ManiR_Limit_Dn,
		bHome_Sensor=> I_ManiR_Limit_Home,
		bBeamAtRight=> I_ManiR_Turned_Right,
		bBeamAtLeft=> I_ManiR_Turned_Left);

	(*Call drill machine*)
	fbDrill(
		bEnable:= bDrill_axZ_Enable,
		bLift_Start:= bDrill_axZ_Start,
		fLift_Velo:= fDrill_axZ_Velo,
		fLift_TargetPos:= fDrill_axZ_TargetPos,
		bDrillOn:= O_Drill_Spindle_On,
		bFixture_Close:= O_Drill_Fixture_Close,
		stPart_inFixture:= stPart_inDrillFixture,
		bLift_InTarget=> bDrill_axZ_InTargetPos,
		fLift_CurrentPos=> fDrill_axZ_CurrPos,
		bLimit_Top=> I_Drill_Limit_Up,
		bLimit_Bottom=> I_Drill_Limit_Dn,
		bHome_Sensor=> I_Drill_Limit_Home,
		bFixture_Open=> I_Drill_Fixture_Open,
		bFixture_Closed=> I_Drill_Fixture_Closed);
END_IF;


(*Make part exchange and check error conditions between ConvIn and ManipLeft*)
ErrorCheck_ManipLeft_ConvIn;
(*Make part exchange and check error conditions between ManipLeft and Drill*)
ErrorCheck_ManipLeft_Drill;
(*Make drilling and check error conditions at Drilling*)
ErrorCheck_Drill;
(*Make part exchange and check error conditions between ManipRight and Drill*)
ErrorCheck_ManipRight_Drill;
(*Make part exchange and check error conditions between ManipRight and ConvOut*)
ErrorCheck_ManipRight_ConvOut;
(*Collisions between devices*)
ErrorCheck_Collisions;


(*drops part from Manipulator Left*)
IF stPart_inMLeftGripper.bExists AND fbManipLeft.bGripperIsOpen THEN
	stPart_inMLeftGripper.bExists := FALSE;
END_IF;
(*drops part from Manipulator Right*)
IF stPart_inMRightGripper.bExists AND fbManipRight.bGripperIsOpen THEN
	stPart_inMRightGripper.bExists := FALSE;
END_IF;



(*Clear active errors*)
IF bClearErrors THEN
	wError_ManipL := 0;
	wError_Drill := 0;
	wError_ManipR := 0;
END_IF;

(*Remove parts from entire system*)
IF bClearSystem THEN
	(*Clear input & output conveyour from parts*)
	FOR i:= 0 TO 10 DO
		arrParts_ConvIn[i].bExists := FALSE;
		arrParts_ConvOut[i].bExists := FALSE;
	END_FOR;
	(*Clear Manipulators and drill from parts*)
	stPart_inMLeftGripper.bExists := FALSE;
	stPart_inDrillFixture.bExists := FALSE;
	stPart_inMRightGripper.bExists := FALSE;
END_IF;
END_PROGRAM
ACTION ErrorCheck_Collisions:
(*ManipL and Conveyor collision*)
IF (fbManipLeft.fPos_Y > 140) AND (fbManipLeft.fPos_angle < 50) THEN
	wError_ManipL.7 := TRUE;	(*collision with conveyor*)
END_IF;

(*ManipL and Drill collision*)
IF ((fbDrill.fPos_Y + 16) > fbManipLeft.fPos_Y) AND fbManipLeft.fPos_angle > 150 THEN
	wError_ManipL.1 := TRUE;
	wError_Drill.0 := TRUE;
END_IF;

(*ManipR and Drill collision*)
IF ((fbDrill.fPos_Y + 10) > fbManipRight.fPos_Y) AND fbManipRight.fPos_angle < 40 THEN	(* was +16 and <50 *)
	wError_ManipR.1 := TRUE;
	wError_Drill.1 := TRUE;
END_IF;

(*ManipR and Conveyor collision*)
IF (fbManipRight.fPos_Y > 140) AND (fbManipRight.fPos_angle > 150) THEN
	wError_ManipR.7 := TRUE;	(*collision with conveyor*)
END_IF;

(*ManipL and ManipR collision*)
IF (fbManipLeft.fPos_angle > 130) AND (fbManipRight.fPos_angle < 50) AND
  (ABS(fbManipRight.fPos_Y - fbManipLeft.fPos_Y) < 60) THEN
	wError_ManipL.9 := TRUE;	(*collision sidewise with ManipulatorRight*)
	wError_ManipR.9 := TRUE;	(*collision sidewise with ManipulatorLeft*)
END_IF;
END_ACTION
ACTION ErrorCheck_Drill:
(*State model for Drilling.
Includes all associated error conditions and judgements *)

(*Drilling cycle has been initiated, but part is removed somewhere between.*)
IF (iState_IF[5] > 0) AND NOT stPart_inDrillFixture.bExists THEN
	iState_IF[5] := 0;
END_IF;

(*Drilled too long*)
IF stPart_inDrillFixture.bExists AND
  (fbDrill.fPos_Y > (fPOS_DRILL_BIT_TOUCHES + fPART_HOLE_DEPTH_MAX)) THEN
	wError_Drill.2 := TRUE;	(*collision with part and Drill*)
END_IF;


CASE iState_IF[5] OF
0: (* IDLE *)
	IF fbDrill.fPos_Y > ( fPOS_DRILL_BIT_TOUCHES - fPART_HEIGH ) THEN
		iState_IF[5] := 1;
	END_IF;

1: (* Approaches with Drill *)
	IF  fbDrill.fPos_Y >= fPOS_DRILL_BIT_TOUCHES THEN
		iState_IF[5] := 2;
	END_IF;

2: (* Drilling *)
	IF fbDrill.fPos_Y >= (fPOS_DRILL_BIT_TOUCHES + fPART_HOLE_DEPTH_REQ ) THEN
		iState_IF[5] := 3;
	END_IF;
	IF stPart_inDrillFixture.bExists AND NOT fbDrill.bFixture_Closed THEN
		wError_Drill.7 := TRUE;	(*Drilling without closed fixture*)
	END_IF;
	IF stPart_inDrillFixture.bExists AND fbDrill.iRPMCurrent < iDRILL_SPINDLE_MIN_FOR_DRILLING THEN
		wError_Drill.2 := TRUE;	(*collision with part and Drill*)
		wError_Drill.6 := TRUE;	(*Drilling without sufficient spindle RPM*)
	END_IF;

3: (* Drilled *)
	stPart_inDrillFixture.bHasHole := TRUE;
	IF fbDrill.fPos_Y < fPOS_DRILL_BIT_TOUCHES THEN
		iState_IF[5] := 4;
	END_IF;

4: (* moved up from part *)
	stPart_inDrillFixture.bHasHole := TRUE;
	IF fbDrill.fPos_Y < 30 THEN
		iState_IF[5] := 5;
	END_IF;

5: (* moved to wait area *)
	iState_IF[5] := 0;

ELSE
	iState_IF[5] := 0;
END_CASE;
END_ACTION
ACTION ErrorCheck_ManipLeft_ConvIn:
(*State model for exchanging part from ConveyorIn to ManipLeft.
Includes all associated error conditions and judgements *)

CASE iState_IF[1] OF
0: (* IDLE *)
	IF arrParts_ConvIn[0].bExists AND NOT stPart_inMLeftGripper.bExists THEN
		iState_IF[1] := 1;
	END_IF;

1: (* waitMoveAbove *)
	IF fbManipLeft.bBeamAtLeft AND fbManipLeft.fPos_Y < fPOS_MANIP_CONV_NO_PART_SAFE THEN
		iState_IF[1] := 2;
	END_IF;
	IF fbManipLeft.fPos_angle < 30 AND fbManipLeft.fPos_Y > fPOS_MANIP_CONV_NO_PART_SAFE THEN
		wError_ManipL.0 := TRUE;
	END_IF;

2: (* ManipulatorLeft is above *)
	IF fbManipLeft.bBeamAtLeft AND fbManipLeft.fPos_Y >= fPOS_MANIP_CONV_NO_PART_SAFE THEN
		iState_IF[1] := 3;
	END_IF;
	IF NOT fbManipLeft.bBeamAtLeft AND fbManipLeft.fPos_angle < 30 AND fbManipLeft.fPos_Y > fPOS_MANIP_CONV_NO_PART_SAFE THEN
		wError_ManipL.0 := TRUE;
	END_IF;

3: (* Approaches from above *)
	IF fbManipLeft.bBeamAtLeft AND fbManipLeft.bGripperIsOpen AND
	  fbManipLeft.fPos_Y >= (fPOS_MANIP_CONV_PICK_LEVEL - 2*fPART_PICK_TOLERANCE) THEN
		iState_IF[1] := 4;
	ELSIF fbManipLeft.fPos_Y < fPOS_MANIP_CONV_NO_PART_SAFE THEN
		iState_IF[1] := 0;
	END_IF;
	IF NOT fbManipLeft.bBeamAtLeft THEN
		wError_ManipL.0 := TRUE;
	END_IF;
	IF NOT fbManipLeft.bGripperIsOpen THEN
		wError_ManipL.5 := TRUE;
	END_IF;

4: (* Over part *)
	IF fbManipLeft.bBeamAtLeft AND fbManipLeft.fPos_Y >= (fPOS_MANIP_CONV_PICK_LEVEL - fPART_PICK_TOLERANCE) AND
	fbManipLeft.fPos_Y <= fPOS_MANIP_CONV_PICK_LEVEL AND fbManipLeft.bGripperClosed THEN
		(*Grasping occurs*)
		iState_IF[1] := 5;
		(*TODO: Add part grasp height compensation*)
	ELSIF fbManipLeft.fPos_Y < fPOS_MANIP_CONV_NO_PART_SAFE THEN
		iState_IF[1] := 0;
	END_IF;
	IF NOT fbManipLeft.bBeamAtLeft THEN
		wError_ManipL.0 := TRUE;
	END_IF;
	IF fbManipLeft.fPos_Y > fPOS_MANIP_CONV_PICK_LEVEL THEN
		wError_ManipL.2 := TRUE;
	END_IF;

5: (* part grasped *)
	stPart_inMLeftGripper.bExists := TRUE;
	IF fbManipLeft.bBeamAtLeft AND fbManipLeft.fPos_Y < fPOS_MANIP_CONV_WITH_PART_SAFE THEN
		iState_IF[1] := 6;
	END_IF;
	IF NOT fbManipLeft.bBeamAtLeft AND fbManipLeft.fPos_Y > fPOS_MANIP_CONV_NO_PART_SAFE THEN
		wError_ManipL.3 := TRUE;
	END_IF;

6: (* moved up with part *)
	IF fbManipLeft.fPos_Y < fPOS_MANIP_CONV_WITH_PART_SAFE THEN
		iState_IF[1] := 7;
	END_IF;

7: (* moved up with part *)
	arrParts_ConvIn[0].bExists := FALSE;
	iState_IF[1] := 0;

ELSE
	iState_IF[1] := 0;
END_CASE;
END_ACTION
ACTION ErrorCheck_ManipLeft_Drill:
(*State model for exchanging part from ManipLeft to Drill.
Includes all associated error conditions and judgements *)

(*Dropping part from gripper too soon*)
IF (iState_IF[2] > 0) AND (iState_IF[2] <= 3) AND NOT fbManipLeft.bGripperClosed AND stPart_inMLeftGripper.bExists THEN
	wError_ManipL.6 := TRUE;
	iState_IF[2] := 0;
END_IF;

(*Collision with parts*)
IF stPart_inMLeftGripper.bExists AND stPart_inDrillFixture.bExists AND fbManipLeft.bBeamAtRight AND
  fbManipLeft.fPos_Y > (fPOS_MANIP_DRILL_PICK_LEVEL - 2* fPART_HEIGH) THEN
	wError_Drill.3 := TRUE;
END_IF;

(*Part exchange sequence*)
CASE iState_IF[2] OF
0: (* IDLE *)
	IF stPart_inMLeftGripper.bExists AND fbManipLeft.bGripperClosed THEN
		iState_IF[2] := 1;
	END_IF;

1: (* waitMoveAbove *)
	IF fbManipLeft.bBeamAtRight AND fbManipLeft.fPos_Y < fPOS_MANIP_DRILL_WITH_PART_SAFE THEN
		iState_IF[2] := 2;
	END_IF;
	IF fbManipLeft.fPos_angle > 150 AND fbManipLeft.fPos_Y > fPOS_MANIP_DRILL_WITH_PART_SAFE THEN
		wError_ManipL.1 := TRUE;
	END_IF;

2: (* ManipulatorLeft is above release point*)
	IF fbManipLeft.bBeamAtRight AND fbManipLeft.fPos_Y >= fPOS_MANIP_DRILL_WITH_PART_SAFE THEN
		iState_IF[2] := 3;
	END_IF;
	IF NOT fbManipLeft.bBeamAtRight AND (fbManipLeft.fPos_angle > 150) AND
	  (fbManipLeft.fPos_Y > fPOS_MANIP_DRILL_WITH_PART_SAFE) THEN
		wError_ManipL.1 := TRUE;
	END_IF;

3: (* Approaches from above *)
	IF fbManipLeft.bBeamAtRight AND fbManipLeft.bGripperClosed AND
	  (fbManipLeft.fPos_Y >= (fPOS_MANIP_DRILL_PICK_LEVEL - fPART_PICK_TOLERANCE)) THEN
		iState_IF[2] := 4;
	ELSIF fbManipLeft.fPos_Y < fPOS_MANIP_DRILL_WITH_PART_SAFE THEN
		iState_IF[2] := 0;
	END_IF;
	IF NOT fbManipLeft.bBeamAtRight AND fbManipLeft.fPos_Y > fPOS_MANIP_DRILL_WITH_PART_SAFE THEN
		wError_ManipL.1 := TRUE;
	END_IF;

4: (* At release point *)
	(*Errors*)
	IF stPart_inDrillFixture.bExists THEN
		wError_ManipL.2 := TRUE;
		wError_Drill.3 := TRUE;
	END_IF;
	(*State trensition*)
	IF fbManipLeft.bBeamAtRight AND (fbManipLeft.fPos_Y >= (fPOS_MANIP_DRILL_PICK_LEVEL - fPART_PICK_TOLERANCE)) AND
	fbManipLeft.fPos_Y <= fPOS_MANIP_DRILL_PICK_LEVEL AND fbManipLeft.bGripperIsOpen THEN
		(*Release occurs*)
		iState_IF[2] := 5;
		(*Copy part to Drill Fixture*)
		F_CopyPart(stPart_inMLeftGripper, stPart_inDrillFixture);
		stPart_inMLeftGripper.bExists := FALSE;
	ELSIF fbManipLeft.fPos_Y < fPOS_MANIP_DRILL_WITH_PART_SAFE THEN
		iState_IF[2] := 0;
	END_IF;
	IF NOT fbManipLeft.bBeamAtRight AND fbManipLeft.fPos_Y > fPOS_MANIP_DRILL_WITH_PART_SAFE THEN
		wError_ManipL.1 := TRUE;
	END_IF;
	IF fbManipLeft.fPos_Y > fPOS_MANIP_DRILL_PICK_LEVEL THEN
		wError_ManipL.2 := TRUE;
	END_IF;
	IF fbDrill.bFixture_Closed THEN
		wError_Drill.4 := TRUE;	(*Fixture closed when inserting part*)
	END_IF;

5: (* Release part *)
	IF fbManipLeft.bBeamAtRight AND fbManipLeft.fPos_Y <= fPOS_MANIP_DRILL_NO_PART_SAFE THEN
		iState_IF[2] := 6;
	ELSIF fbManipLeft.bBeamAtLeft AND fbManipLeft.fPos_Y <= fPOS_MANIP_CONV_NO_PART_SAFE THEN
		(* Errornous leave condition*)
		iState_IF[2] := 0;
	END_IF;
	IF NOT fbManipLeft.bBeamAtRight AND fbManipLeft.fPos_Y > fPOS_MANIP_DRILL_NO_PART_SAFE THEN
		wError_ManipL.1 := TRUE;
		wError_ManipL.3 := TRUE;
	END_IF;
	IF NOT fbManipLeft.bGripperIsOpen THEN
		wError_ManipR.10 := TRUE;	(*re-grasping released part*)
	END_IF;

6: (* moved up *)
	IF fbManipLeft.fPos_Y <= fPOS_MANIP_DRILL_NO_PART_SAFE THEN
		iState_IF[2] := 7;
	END_IF;
	iState_IF[2] := 0;

7: (* Can move away *)
	iState_IF[2] := 0;

ELSE
	iState_IF[2] := 0;
END_CASE;
END_ACTION
ACTION ErrorCheck_ManipRight_ConvOut:
(*State model for exchanging part from ManipRight to Conveyor.
Includes all associated error conditions and judgements *)

(*Dropping part from gripper too soon*)
IF (iState_IF[4] > 0) AND (iState_IF[4] <= 3) AND NOT fbManipRight.bGripperClosed AND stPart_inMRightGripper.bExists THEN
	wError_ManipR.6 := TRUE;
	iState_IF[4] := 0;
END_IF;

(*Collision with parts*)
IF stPart_inMRightGripper.bExists AND arrParts_ConvOut[5].bExists AND fbManipRight.fPos_angle > 150 AND
  fbManipRight.fPos_Y > (fPOS_MANIP_CONV_PICK_LEVEL - fPART_HEIGH) THEN
	wError_ManipR.8 := TRUE;
END_IF;

(*Part exchange sequence*)
CASE iState_IF[4] OF
0: (* IDLE *)
	IF stPart_inMRightGripper.bExists AND fbManipRight.bGripperClosed THEN
		iState_IF[4] := 1;
	END_IF;

1: (* waitMoveAbove *)
	IF fbManipRight.bBeamAtRight AND fbManipRight.fPos_Y <= fPOS_MANIP_CONV_WITH_PART_SAFE THEN
		iState_IF[4] := 2;
	END_IF;
	IF fbManipRight.fPos_angle > 150 AND fbManipRight.fPos_Y > fPOS_MANIP_CONV_WITH_PART_SAFE THEN
		wError_ManipR.0 := TRUE;
	END_IF;

2: (* ManipulatorRight is above release point*)
	IF fbManipRight.bBeamAtRight AND fbManipRight.fPos_Y >= fPOS_MANIP_CONV_WITH_PART_SAFE THEN
		iState_IF[4] := 3;
	END_IF;
	IF NOT fbManipRight.bBeamAtRight AND (fbManipRight.fPos_angle > 150) AND
	  (fbManipRight.fPos_Y > fPOS_MANIP_CONV_WITH_PART_SAFE) THEN
		wError_ManipR.0 := TRUE;
	END_IF;

3: (* Approaches from above *)
	IF fbManipRight.bBeamAtRight AND fbManipRight.bGripperClosed AND
	  (fbManipRight.fPos_Y >= (fPOS_MANIP_CONV_PICK_LEVEL - fPART_PICK_TOLERANCE)) THEN
		iState_IF[4] := 4;
	ELSIF fbManipRight.fPos_Y < fPOS_MANIP_CONV_WITH_PART_SAFE THEN
		iState_IF[4] := 0;
	END_IF;
	IF NOT fbManipRight.bBeamAtRight AND fbManipRight.fPos_Y > fPOS_MANIP_CONV_WITH_PART_SAFE THEN
		wError_ManipR.0 := TRUE;
	END_IF;

4: (* At release point *)
	(*Errors*)
	IF arrParts_ConvOut[5].bExists THEN
		wError_ManipR.2 := TRUE;
	END_IF;
	(*State trensition*)
	IF fbManipRight.bBeamAtRight AND (fbManipRight.fPos_Y >= (fPOS_MANIP_CONV_PICK_LEVEL - fPART_PICK_TOLERANCE)) AND
	fbManipRight.fPos_Y <= fPOS_MANIP_CONV_PICK_LEVEL AND fbManipRight.bGripperIsOpen THEN
		(*Release occurs*)
		iState_IF[4] := 5;
		(*Copy part to Conveyour Out*)
		F_CopyPart(stPart_inMRightGripper, arrParts_ConvOut[5]);
		(*TODO: Add part grasp height compensation*)
	ELSIF fbManipRight.fPos_Y < fPOS_MANIP_CONV_WITH_PART_SAFE THEN
		iState_IF[4] := 0;
	END_IF;
	IF NOT fbManipRight.bBeamAtRight AND fbManipRight.fPos_Y > fPOS_MANIP_CONV_WITH_PART_SAFE THEN
		wError_ManipR.1 := TRUE;
	END_IF;
	IF fbManipRight.fPos_Y > fPOS_MANIP_CONV_PICK_LEVEL THEN
		wError_ManipR.2 := TRUE;
	END_IF;

5: (* Release part *)
	stPart_inMRightGripper.bExists := FALSE;
	IF fbManipRight.bBeamAtRight AND fbManipRight.fPos_Y <= fPOS_MANIP_CONV_NO_PART_SAFE AND
	   fbManipRight.bGripperIsOpen THEN
		iState_IF[4] := 6;
	END_IF;
	IF NOT fbManipRight.bBeamAtRight AND fbManipRight.fPos_Y > fPOS_MANIP_CONV_NO_PART_SAFE THEN
		wError_ManipR.1 := TRUE;
		wError_ManipR.3 := TRUE;
	END_IF;
	IF NOT fbManipRight.bGripperIsOpen THEN
		wError_ManipR.10 := TRUE;	(*re-grasping released part*)
	END_IF;

6: (* moved up *)
	iState_IF[4] := 0;

ELSE
	iState_IF[4] := 0;
END_CASE;
END_ACTION
ACTION ErrorCheck_ManipRight_Drill:
(*State model for exchanging part from Drive to ManipRight.
Includes all associated error conditions and judgements *)

CASE iState_IF[3] OF
0: (* IDLE *)
	IF stPart_inDrillFixture.bExists AND NOT stPart_inMRightGripper.bExists THEN
		iState_IF[3] := 1;
	END_IF;

1: (* waitMoveAbove *)
	IF fbManipRight.bBeamAtLeft AND fbManipRight.fPos_Y <= fPOS_MANIP_DRILL_NO_PART_SAFE THEN
		iState_IF[3] := 2;
	END_IF;
	IF fbManipRight.fPos_angle < 30 AND fbManipRight.fPos_Y > fPOS_MANIP_DRILL_NO_PART_SAFE THEN
		wError_ManipR.1 := TRUE;
	END_IF;

2: (* ManipulatorLeft is above *)
	IF fbManipRight.bBeamAtLeft AND fbManipRight.fPos_Y >= fPOS_MANIP_DRILL_NO_PART_SAFE THEN
		iState_IF[3] := 3;
	END_IF;
	IF NOT fbManipRight.bBeamAtLeft AND fbManipRight.fPos_angle > 30 AND fbManipRight.fPos_Y > fPOS_MANIP_DRILL_NO_PART_SAFE THEN
		wError_ManipR.1 := TRUE;
	END_IF;

3: (* Approaches from above *)
	IF fbManipRight.bBeamAtLeft AND fbManipRight.bGripperIsOpen AND
	  fbManipRight.fPos_Y >= (fPOS_MANIP_DRILL_PICK_LEVEL - fPART_PICK_TOLERANCE) THEN
		iState_IF[3] := 4;
	ELSIF fbManipRight.fPos_Y < fPOS_MANIP_DRILL_NO_PART_SAFE THEN
		iState_IF[3] := 0;
	END_IF;
	IF NOT fbManipRight.bBeamAtLeft THEN
		wError_ManipR.1 := TRUE;
	END_IF;
	IF NOT fbManipRight.bGripperIsOpen THEN
		wError_ManipR.5 := TRUE;
	END_IF;

